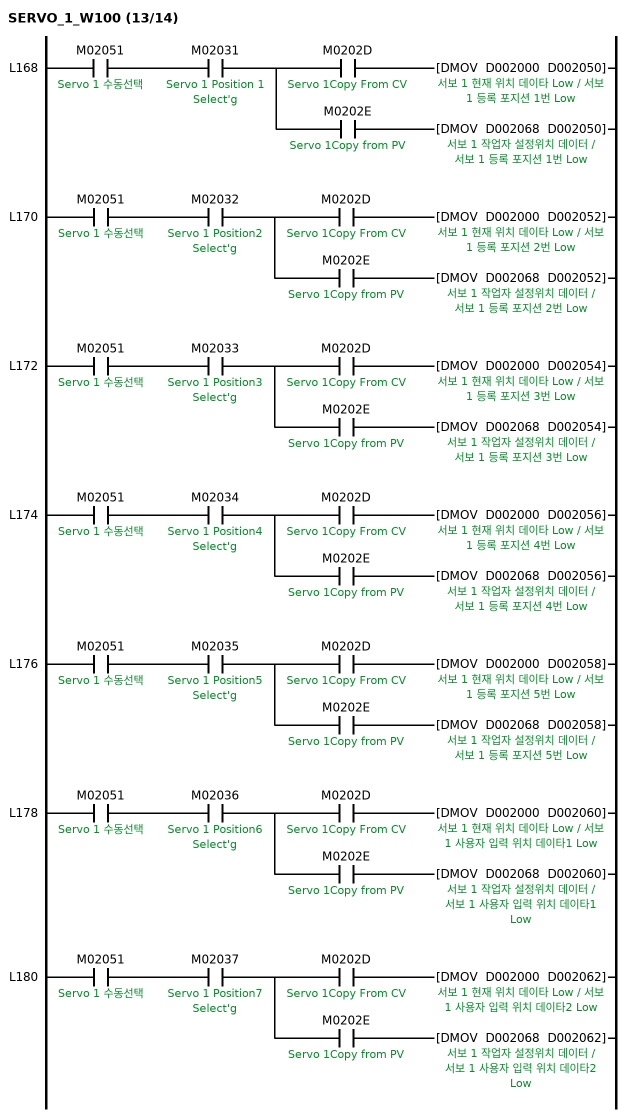
[picture p288: SERVO_1_W100 rungs L168-L180]
; L168
LOAD      M02051	// Servo 1 수동선택
AND       M02031	// Servo 1 Position 1 Select'g
MPUSH
AND       M0202D	// Servo 1Copy From CV
DMOV      D002000 D002050	// 서보 1 현재 위치 데이타 Low / 서보 1 등록 포지션 1번 Low
MPOP
AND       M0202E	// Servo 1Copy from PV
DMOV      D002068 D002050	// 서보 1 작업자 설정위치 데이터 / 서보 1 등록 포지션 1번 Low
; L170
LOAD      M02051	// Servo 1 수동선택
AND       M02032	// Servo 1 Position2 Select'g
MPUSH
AND       M0202D	// Servo 1Copy From CV
DMOV      D002000 D002052	// 서보 1 현재 위치 데이타 Low / 서보 1 등록 포지션 2번 Low
MPOP
AND       M0202E	// Servo 1Copy from PV
DMOV      D002068 D002052	// 서보 1 작업자 설정위치 데이터 / 서보 1 등록 포지션 2번 Low
; L172
LOAD      M02051	// Servo 1 수동선택
AND       M02033	// Servo 1 Position3 Select'g
MPUSH
AND       M0202D	// Servo 1Copy From CV
DMOV      D002000 D002054	// 서보 1 현재 위치 데이타 Low / 서보 1 등록 포지션 3번 Low
MPOP
AND       M0202E	// Servo 1Copy from PV
DMOV      D002068 D002054	// 서보 1 작업자 설정위치 데이터 / 서보 1 등록 포지션 3번 Low
; L174
LOAD      M02051	// Servo 1 수동선택
AND       M02034	// Servo 1 Position4 Select'g
MPUSH
AND       M0202D	// Servo 1Copy From CV
DMOV      D002000 D002056	// 서보 1 현재 위치 데이타 Low / 서보 1 등록 포지션 4번 Low
MPOP
AND       M0202E	// Servo 1Copy from PV
DMOV      D002068 D002056	// 서보 1 작업자 설정위치 데이터 / 서보 1 등록 포지션 4번 Low
; L176
LOAD      M02051	// Servo 1 수동선택
AND       M02035	// Servo 1 Position5 Select'g
MPUSH
AND       M0202D	// Servo 1Copy From CV
DMOV      D002000 D002058	// 서보 1 현재 위치 데이타 Low / 서보 1 등록 포지션 5번 Low
MPOP
AND       M0202E	// Servo 1Copy from PV
DMOV      D002068 D002058	// 서보 1 작업자 설정위치 데이터 / 서보 1 등록 포지션 5번 Low
; L178
LOAD      M02051	// Servo 1 수동선택
AND       M02036	// Servo 1 Position6 Select'g
MPUSH
AND       M0202D	// Servo 1Copy From CV
DMOV      D002000 D002060	// 서보 1 현재 위치 데이타 Low / 서보 1 사용자 입력 위치 데이타1 Low
MPOP
AND       M0202E	// Servo 1Copy from PV
DMOV      D002068 D002060	// 서보 1 작업자 설정위치 데이터 / 서보 1 사용자 입력 위치 데이타1 Low
; L180
LOAD      M02051	// Servo 1 수동선택
AND       M02037	// Servo 1 Position7 Select'g
MPUSH
AND       M0202D	// Servo 1Copy From CV
DMOV      D002000 D002062	// 서보 1 현재 위치 데이타 Low / 서보 1 사용자 입력 위치 데이타2 Low
MPOP
AND       M0202E	// Servo 1Copy from PV
DMOV      D002068 D002062	// 서보 1 작업자 설정위치 데이터 / 서보 1 사용자 입력 위치 데이타2 Low

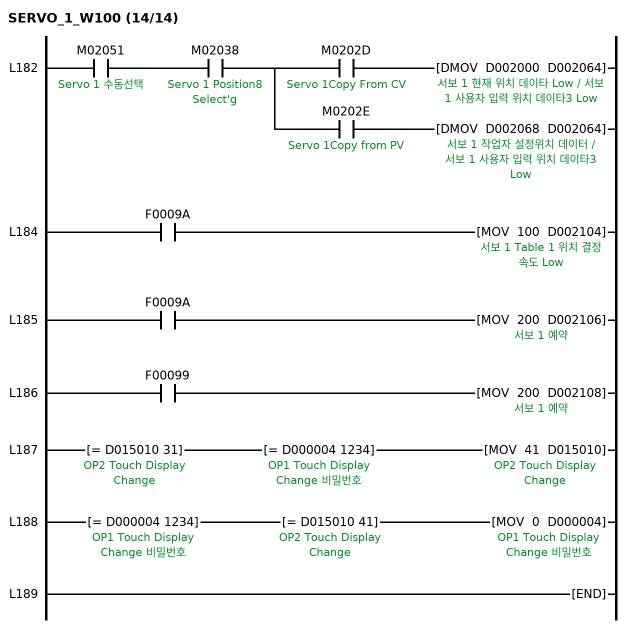
; L182
LOAD      M02051	// Servo 1 수동선택
AND       M02038	// Servo 1 Position8 Select'g
MPUSH
AND       M0202D	// Servo 1Copy From CV
DMOV      D002000 D002064	// 서보 1 현재 위치 데이타 Low / 서보 1 사용자 입력 위치 데이타3 Low
MPOP
AND       M0202E	// Servo 1Copy from PV
DMOV      D002068 D002064	// 서보 1 작업자 설정위치 데이터 / 서보 1 사용자 입력 위치 데이타3 Low
; L184
LOAD      F0009A
MOV       100 D002104	// 서보 1 Table 1 위치 결정 속도 Low
; L185
LOAD      F0009A
MOV       200 D002106	// 서보 1 예약
; L186
LOAD      F00099
MOV       200 D002108	// 서보 1 예약
; L187
LOAD=     D015010 31	// OP2 Touch Display Change
AND=      D000004 1234	// OP1 Touch Display Change 비밀번호
MOV       41 D015010	// OP2 Touch Display Change
; L188
LOAD=     D000004 1234	// OP1 Touch Display Change 비밀번호
AND=      D015010 41	// OP2 Touch Display Change
MOV       0 D000004	// OP1 Touch Display Change 비밀번호
; L189
END

PROGRAM SERVO_2_W200 (task: 스캔 프로그램)

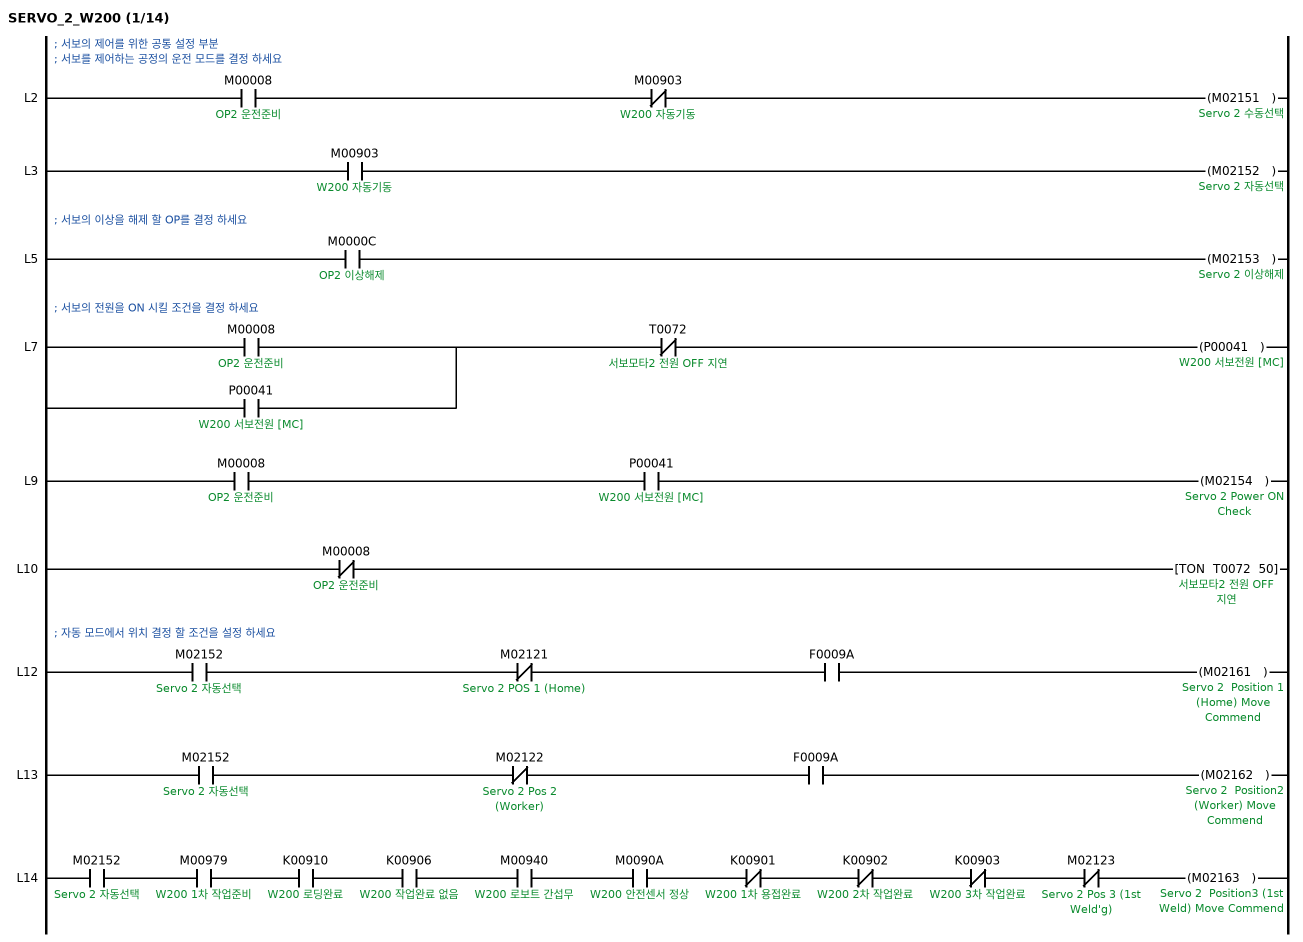
// 서보의 제어를 위한 공통 설정 부분
//     서보를 제어하는 공정의 운전 모드를 결정 하세요
; L2
LOAD      M00008	// OP2 운전준비
AND NOT   M00903	// W200 자동기동
OUT       M02151	// Servo 2 수동선택
; L3
LOAD      M00903	// W200 자동기동
OUT       M02152	// Servo 2 자동선택
//     서보의 이상을 해제 할 OP를 결정 하세요
; L5
LOAD      M0000C	// OP2 이상해제
OUT       M02153	// Servo 2 이상해제
//     서보의 전원을 ON 시킬 조건을 결정 하세요
; L7
LOAD      M00008	// OP2 운전준비
OR        P00041	// W200 서보전원 [MC]
AND NOT   T0072	// 서보모타2 전원 OFF 지연
OUT       P00041	// W200 서보전원 [MC]
; L9
LOAD      M00008	// OP2 운전준비
AND       P00041	// W200 서보전원 [MC]
OUT       M02154	// Servo 2 Power ON Check
; L10
LOAD NOT  M00008	// OP2 운전준비
TON       T0072 50	// 서보모타2 전원 OFF 지연
//     자동 모드에서 위치 결정 할 조건을 설정 하세요
; L12
LOAD      M02152	// Servo 2 자동선택
AND NOT   M02121	// Servo 2 POS 1 (Home)
AND       F0009A
OUT       M02161	// Servo 2  Position 1 (Home) Move Commend
; L13
LOAD      M02152	// Servo 2 자동선택
AND NOT   M02122	// Servo 2 Pos 2 (Worker)
AND       F0009A
OUT       M02162	// Servo 2  Position2 (Worker) Move Commend
; L14
LOAD      M02152	// Servo 2 자동선택
AND       M00979	// W200 1차 작업준비
AND       K00910	// W200 로딩완료
AND       K00906	// W200 작업완료 없음
AND       M00940	// W200 로보트 간섭무
AND       M0090A	// W200 안전센서 정상
AND NOT   K00901	// W200 1차 용접완료
AND NOT   K00902	// W200 2차 작업완료
AND NOT   K00903	// W200 3차 작업완료
AND NOT   M02123	// Servo 2 Pos 3 (1st Weld'g)
OUT       M02163	// Servo 2  Position3 (1st Weld) Move Commend

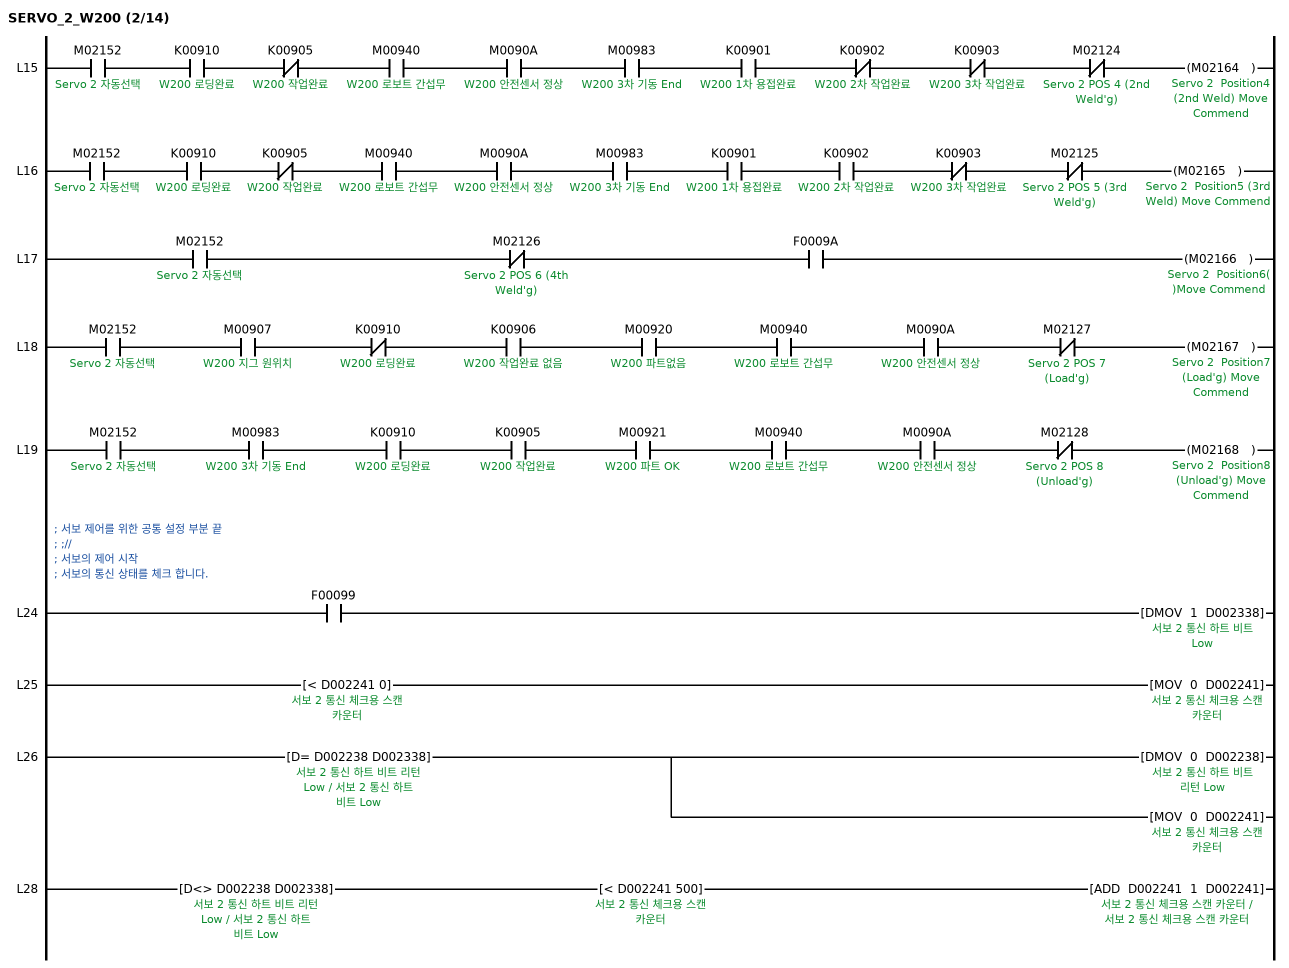
; L15
LOAD      M02152	// Servo 2 자동선택
AND       K00910	// W200 로딩완료
AND NOT   K00905	// W200 작업완료
AND       M00940	// W200 로보트 간섭무
AND       M0090A	// W200 안전센서 정상
AND       M00983	// W200 3차 기동 End
AND       K00901	// W200 1차 용접완료
AND NOT   K00902	// W200 2차 작업완료
AND NOT   K00903	// W200 3차 작업완료
AND NOT   M02124	// Servo 2 POS 4 (2nd Weld'g)
OUT       M02164	// Servo 2  Position4 (2nd Weld) Move Commend
; L16
LOAD      M02152	// Servo 2 자동선택
AND       K00910	// W200 로딩완료
AND NOT   K00905	// W200 작업완료
AND       M00940	// W200 로보트 간섭무
AND       M0090A	// W200 안전센서 정상
AND       M00983	// W200 3차 기동 End
AND       K00901	// W200 1차 용접완료
AND       K00902	// W200 2차 작업완료
AND NOT   K00903	// W200 3차 작업완료
AND NOT   M02125	// Servo 2 POS 5 (3rd Weld'g)
OUT       M02165	// Servo 2  Position5 (3rd Weld) Move Commend
; L17
LOAD      M02152	// Servo 2 자동선택
AND NOT   M02126	// Servo 2 POS 6 (4th Weld'g)
AND       F0009A
OUT       M02166	// Servo 2  Position6()Move Commend
; L18
LOAD      M02152	// Servo 2 자동선택
AND       M00907	// W200 지그 원위치
AND NOT   K00910	// W200 로딩완료
AND       K00906	// W200 작업완료 없음
AND       M00920	// W200 파트없음
AND       M00940	// W200 로보트 간섭무
AND       M0090A	// W200 안전센서 정상
AND NOT   M02127	// Servo 2 POS 7 (Load'g)
OUT       M02167	// Servo 2  Position7 (Load'g) Move Commend
; L19
LOAD      M02152	// Servo 2 자동선택
AND       M00983	// W200 3차 기동 End
AND       K00910	// W200 로딩완료
AND       K00905	// W200 작업완료
AND       M00921	// W200 파트 OK
AND       M00940	// W200 로보트 간섭무
AND       M0090A	// W200 안전센서 정상
AND NOT   M02128	// Servo 2 POS 8 (Unload'g)
OUT       M02168	// Servo 2  Position8 (Unload'g) Move Commend
// 서보 제어를 위한 공통 설정 부분 끝
// ;//
// 서보의 제어 시작
//     서보의 통신 상태를 체크 합니다.
; L24
LOAD      F00099
DMOV      1 D002338	// 서보 2 통신 하트 비트 Low
; L25
LOAD<     D002241 0	// 서보 2 통신 체크용 스캔 카운터
MOV       0 D002241	// 서보 2 통신 체크용 스캔 카운터
; L26
LOADD=    D002238 D002338	// 서보 2 통신 하트 비트 리턴 Low / 서보 2 통신 하트 비트 Low
DMOV      0 D002238	// 서보 2 통신 하트 비트 리턴 Low
MOV       0 D002241	// 서보 2 통신 체크용 스캔 카운터
; L28
LOADD<>   D002238 D002338	// 서보 2 통신 하트 비트 리턴 Low / 서보 2 통신 하트 비트 Low
AND<      D002241 500	// 서보 2 통신 체크용 스캔 카운터
ADD       D002241 1 D002241	// 서보 2 통신 체크용 스캔 카운터 / 서보 2 통신 체크용 스캔 카운터

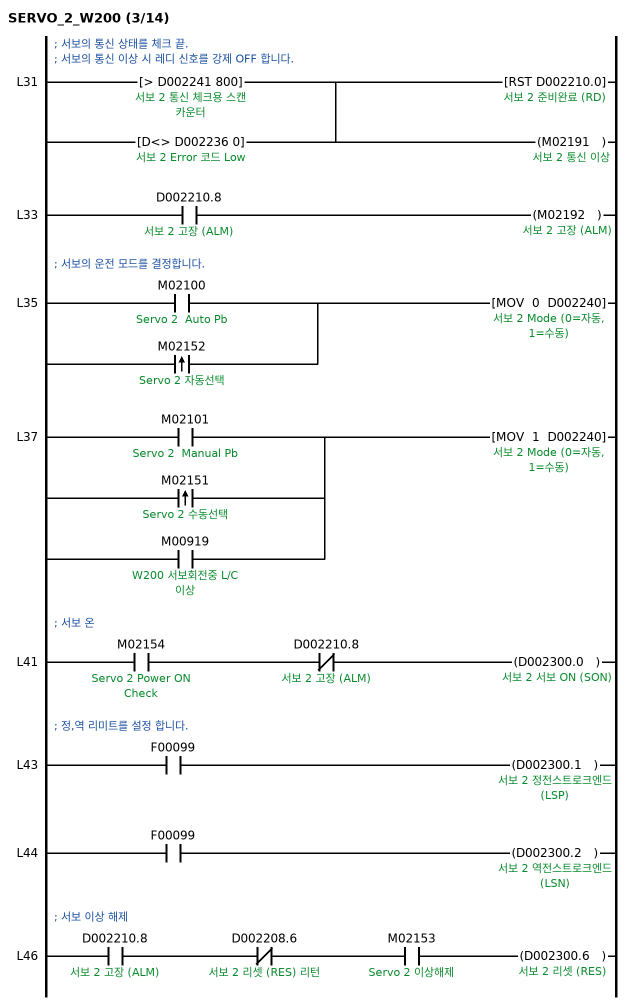
//     서보의 통신 상태를 체크 끝.
//     서보의 통신 이상 시 레디 신호를 강제 OFF 합니다.
; L31
LOAD>     D002241 800	// 서보 2 통신 체크용 스캔 카운터
ORD<>     D002236 0	// 서보 2 Error 코드 Low
RST       D002210.0	// 서보 2 준비완료 (RD)
OUT       M02191	// 서보 2 통신 이상
; L33
LOAD      D002210.8	// 서보 2 고장 (ALM)
OUT       M02192	// 서보 2 고장 (ALM)
//     서보의 운전 모드를 결정합니다.
; L35
LOAD      M02100	// Servo 2  Auto Pb
ORP       M02152	// Servo 2 자동선택
MOV       0 D002240	// 서보 2 Mode (0=자동, 1=수동)
; L37
LOAD      M02101	// Servo 2  Manual Pb
ORP       M02151	// Servo 2 수동선택
OR        M00919	// W200 서보회전중 L/C 이상
MOV       1 D002240	// 서보 2 Mode (0=자동, 1=수동)
//     서보 온
; L41
LOAD      M02154	// Servo 2 Power ON Check
AND NOT   D002210.8	// 서보 2 고장 (ALM)
OUT       D002300.0	// 서보 2 서보 ON (SON)
//     정,역 리미트를 설정 합니다.
; L43
LOAD      F00099
OUT       D002300.1	// 서보 2 정전스트로크엔드 (LSP)
; L44
LOAD      F00099
OUT       D002300.2	// 서보 2 역전스트로크엔드 (LSN)
//     서보 이상 해제
; L46
LOAD      D002210.8	// 서보 2 고장 (ALM)
AND NOT   D002208.6	// 서보 2 리셋 (RES) 리턴
AND       M02153	// Servo 2 이상해제
OUT       D002300.6	// 서보 2 리셋 (RES)

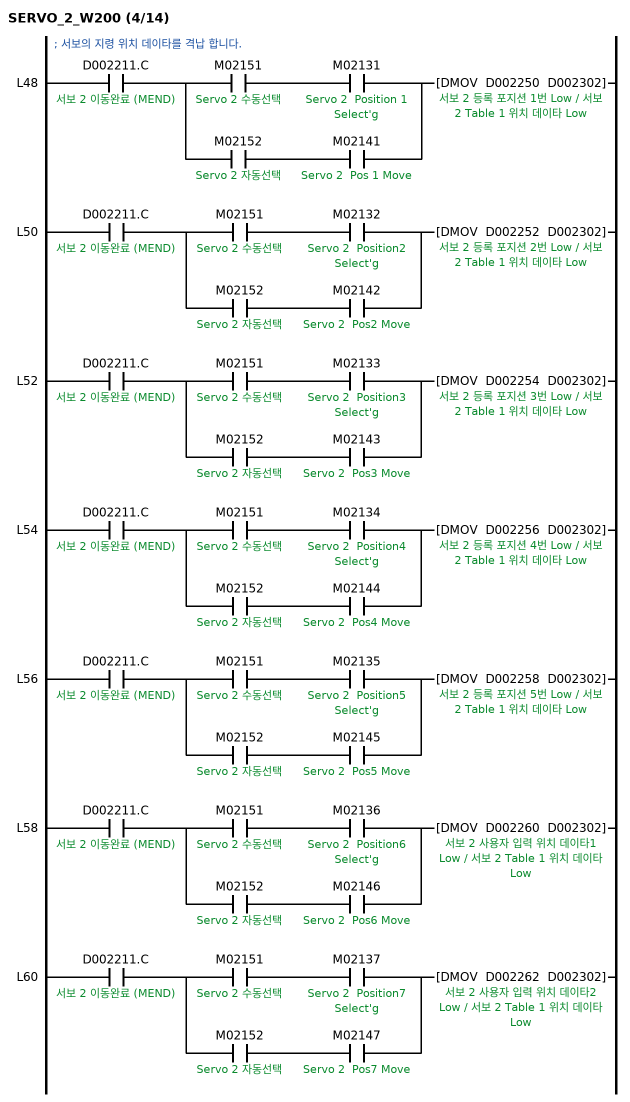
//     서보의 지령 위치 데이타를 격납 합니다.
; L48
LOAD      D002211.C	// 서보 2 이동완료 (MEND)
LOAD      M02151	// Servo 2 수동선택
AND       M02131	// Servo 2  Position 1 Select'g
LOAD      M02152	// Servo 2 자동선택
AND       M02141	// Servo 2  Pos 1 Move
OR LOAD
AND LOAD
DMOV      D002250 D002302	// 서보 2 등록 포지션 1번 Low / 서보 2 Table 1 위치 데이타 Low
; L50
LOAD      D002211.C	// 서보 2 이동완료 (MEND)
LOAD      M02151	// Servo 2 수동선택
AND       M02132	// Servo 2  Position2 Select'g
LOAD      M02152	// Servo 2 자동선택
AND       M02142	// Servo 2  Pos2 Move
OR LOAD
AND LOAD
DMOV      D002252 D002302	// 서보 2 등록 포지션 2번 Low / 서보 2 Table 1 위치 데이타 Low
; L52
LOAD      D002211.C	// 서보 2 이동완료 (MEND)
LOAD      M02151	// Servo 2 수동선택
AND       M02133	// Servo 2  Position3 Select'g
LOAD      M02152	// Servo 2 자동선택
AND       M02143	// Servo 2  Pos3 Move
OR LOAD
AND LOAD
DMOV      D002254 D002302	// 서보 2 등록 포지션 3번 Low / 서보 2 Table 1 위치 데이타 Low
; L54
LOAD      D002211.C	// 서보 2 이동완료 (MEND)
LOAD      M02151	// Servo 2 수동선택
AND       M02134	// Servo 2  Position4 Select'g
LOAD      M02152	// Servo 2 자동선택
AND       M02144	// Servo 2  Pos4 Move
OR LOAD
AND LOAD
DMOV      D002256 D002302	// 서보 2 등록 포지션 4번 Low / 서보 2 Table 1 위치 데이타 Low
; L56
LOAD      D002211.C	// 서보 2 이동완료 (MEND)
LOAD      M02151	// Servo 2 수동선택
AND       M02135	// Servo 2  Position5 Select'g
LOAD      M02152	// Servo 2 자동선택
AND       M02145	// Servo 2  Pos5 Move
OR LOAD
AND LOAD
DMOV      D002258 D002302	// 서보 2 등록 포지션 5번 Low / 서보 2 Table 1 위치 데이타 Low
; L58
LOAD      D002211.C	// 서보 2 이동완료 (MEND)
LOAD      M02151	// Servo 2 수동선택
AND       M02136	// Servo 2  Position6 Select'g
LOAD      M02152	// Servo 2 자동선택
AND       M02146	// Servo 2  Pos6 Move
OR LOAD
AND LOAD
DMOV      D002260 D002302	// 서보 2 사용자 입력 위치 데이타1 Low / 서보 2 Table 1 위치 데이타 Low
; L60
LOAD      D002211.C	// 서보 2 이동완료 (MEND)
LOAD      M02151	// Servo 2 수동선택
AND       M02137	// Servo 2  Position7 Select'g
LOAD      M02152	// Servo 2 자동선택
AND       M02147	// Servo 2  Pos7 Move
OR LOAD
AND LOAD
DMOV      D002262 D002302	// 서보 2 사용자 입력 위치 데이타2 Low / 서보 2 Table 1 위치 데이타 Low

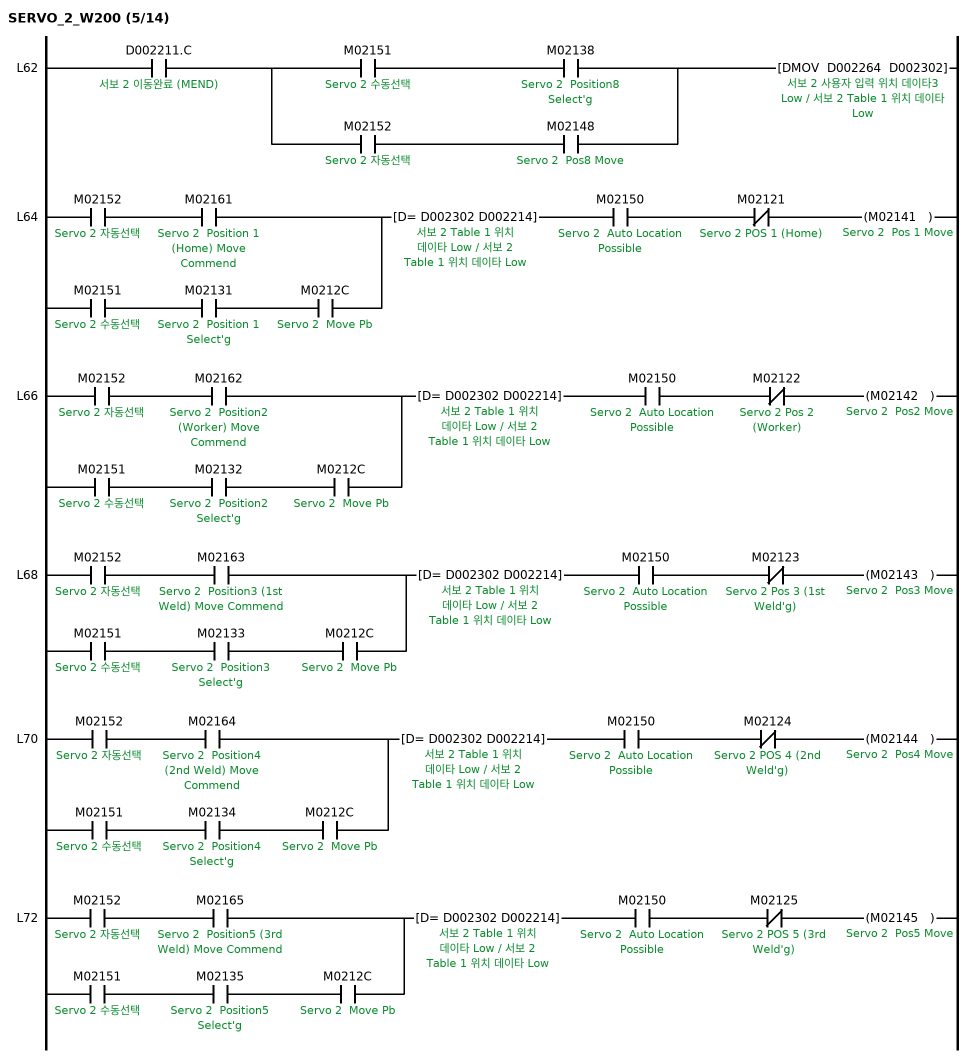
; L62
LOAD      D002211.C	// 서보 2 이동완료 (MEND)
LOAD      M02151	// Servo 2 수동선택
AND       M02138	// Servo 2  Position8 Select'g
LOAD      M02152	// Servo 2 자동선택
AND       M02148	// Servo 2  Pos8 Move
OR LOAD
AND LOAD
DMOV      D002264 D002302	// 서보 2 사용자 입력 위치 데이타3 Low / 서보 2 Table 1 위치 데이타 Low
; L64
LOAD      M02152	// Servo 2 자동선택
AND       M02161	// Servo 2  Position 1 (Home) Move Commend
LOAD      M02151	// Servo 2 수동선택
AND       M02131	// Servo 2  Position 1 Select'g
AND       M0212C	// Servo 2  Move Pb
OR LOAD
ANDD=     D002302 D002214	// 서보 2 Table 1 위치 데이타 Low / 서보 2 Table 1 위치 데이타 Low
AND       M02150	// Servo 2  Auto Location Possible
AND NOT   M02121	// Servo 2 POS 1 (Home)
OUT       M02141	// Servo 2  Pos 1 Move
; L66
LOAD      M02152	// Servo 2 자동선택
AND       M02162	// Servo 2  Position2 (Worker) Move Commend
LOAD      M02151	// Servo 2 수동선택
AND       M02132	// Servo 2  Position2 Select'g
AND       M0212C	// Servo 2  Move Pb
OR LOAD
ANDD=     D002302 D002214	// 서보 2 Table 1 위치 데이타 Low / 서보 2 Table 1 위치 데이타 Low
AND       M02150	// Servo 2  Auto Location Possible
AND NOT   M02122	// Servo 2 Pos 2 (Worker)
OUT       M02142	// Servo 2  Pos2 Move
; L68
LOAD      M02152	// Servo 2 자동선택
AND       M02163	// Servo 2  Position3 (1st Weld) Move Commend
LOAD      M02151	// Servo 2 수동선택
AND       M02133	// Servo 2  Position3 Select'g
AND       M0212C	// Servo 2  Move Pb
OR LOAD
ANDD=     D002302 D002214	// 서보 2 Table 1 위치 데이타 Low / 서보 2 Table 1 위치 데이타 Low
AND       M02150	// Servo 2  Auto Location Possible
AND NOT   M02123	// Servo 2 Pos 3 (1st Weld'g)
OUT       M02143	// Servo 2  Pos3 Move
; L70
LOAD      M02152	// Servo 2 자동선택
AND       M02164	// Servo 2  Position4 (2nd Weld) Move Commend
LOAD      M02151	// Servo 2 수동선택
AND       M02134	// Servo 2  Position4 Select'g
AND       M0212C	// Servo 2  Move Pb
OR LOAD
ANDD=     D002302 D002214	// 서보 2 Table 1 위치 데이타 Low / 서보 2 Table 1 위치 데이타 Low
AND       M02150	// Servo 2  Auto Location Possible
AND NOT   M02124	// Servo 2 POS 4 (2nd Weld'g)
OUT       M02144	// Servo 2  Pos4 Move
; L72
LOAD      M02152	// Servo 2 자동선택
AND       M02165	// Servo 2  Position5 (3rd Weld) Move Commend
LOAD      M02151	// Servo 2 수동선택
AND       M02135	// Servo 2  Position5 Select'g
AND       M0212C	// Servo 2  Move Pb
OR LOAD
ANDD=     D002302 D002214	// 서보 2 Table 1 위치 데이타 Low / 서보 2 Table 1 위치 데이타 Low
AND       M02150	// Servo 2  Auto Location Possible
AND NOT   M02125	// Servo 2 POS 5 (3rd Weld'g)
OUT       M02145	// Servo 2  Pos5 Move

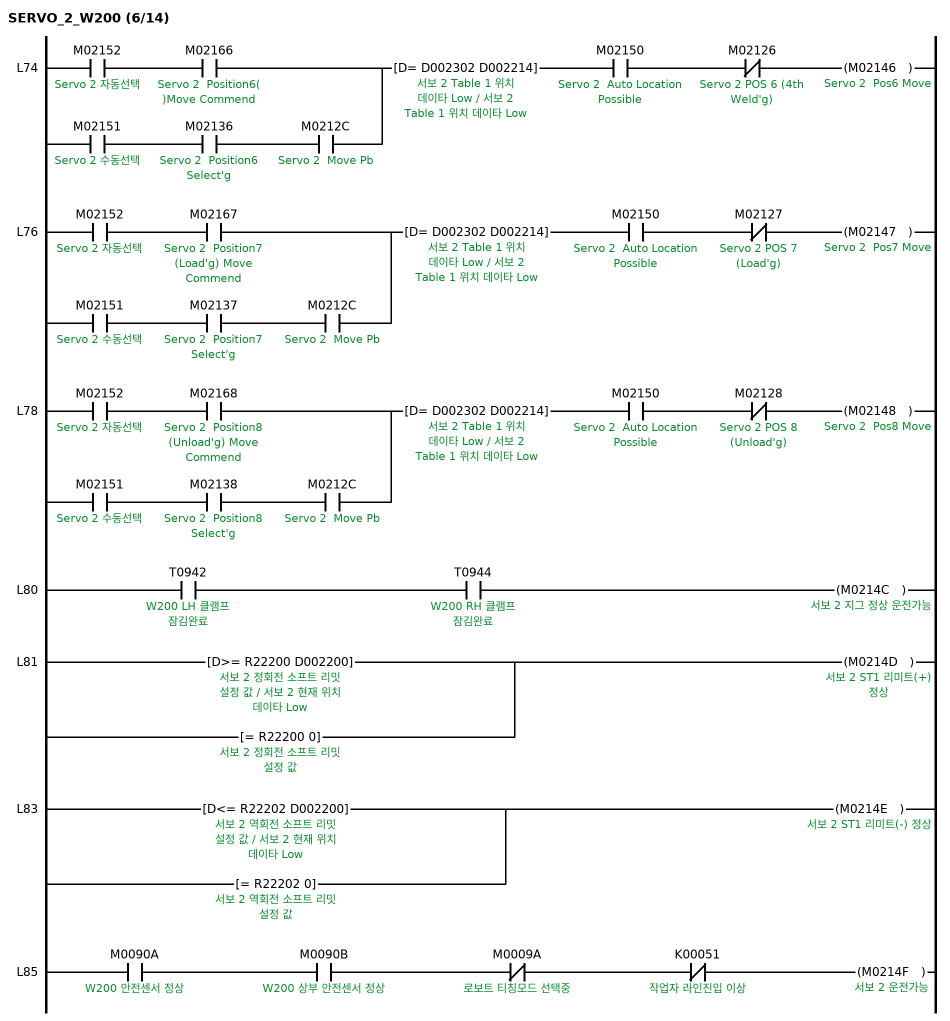
; L74
LOAD      M02152	// Servo 2 자동선택
AND       M02166	// Servo 2  Position6()Move Commend
LOAD      M02151	// Servo 2 수동선택
AND       M02136	// Servo 2  Position6 Select'g
AND       M0212C	// Servo 2  Move Pb
OR LOAD
ANDD=     D002302 D002214	// 서보 2 Table 1 위치 데이타 Low / 서보 2 Table 1 위치 데이타 Low
AND       M02150	// Servo 2  Auto Location Possible
AND NOT   M02126	// Servo 2 POS 6 (4th Weld'g)
OUT       M02146	// Servo 2  Pos6 Move
; L76
LOAD      M02152	// Servo 2 자동선택
AND       M02167	// Servo 2  Position7 (Load'g) Move Commend
LOAD      M02151	// Servo 2 수동선택
AND       M02137	// Servo 2  Position7 Select'g
AND       M0212C	// Servo 2  Move Pb
OR LOAD
ANDD=     D002302 D002214	// 서보 2 Table 1 위치 데이타 Low / 서보 2 Table 1 위치 데이타 Low
AND       M02150	// Servo 2  Auto Location Possible
AND NOT   M02127	// Servo 2 POS 7 (Load'g)
OUT       M02147	// Servo 2  Pos7 Move
; L78
LOAD      M02152	// Servo 2 자동선택
AND       M02168	// Servo 2  Position8 (Unload'g) Move Commend
LOAD      M02151	// Servo 2 수동선택
AND       M02138	// Servo 2  Position8 Select'g
AND       M0212C	// Servo 2  Move Pb
OR LOAD
ANDD=     D002302 D002214	// 서보 2 Table 1 위치 데이타 Low / 서보 2 Table 1 위치 데이타 Low
AND       M02150	// Servo 2  Auto Location Possible
AND NOT   M02128	// Servo 2 POS 8 (Unload'g)
OUT       M02148	// Servo 2  Pos8 Move
; L80
LOAD      T0942	// W200 LH 클램프 잠김완료
AND       T0944	// W200 RH 클램프 잠김완료
OUT       M0214C	// 서보 2 지그 정상 운전가능
; L81
LOADD>=   R22200 D002200	// 서보 2 정회전 소프트 리밋 설정 값 / 서보 2 현재 위치 데이타 Low
OR=       R22200 0	// 서보 2 정회전 소프트 리밋 설정 값
OUT       M0214D	// 서보 2 ST1 리미트(+) 정상
; L83
LOADD<=   R22202 D002200	// 서보 2 역회전 소프트 리밋 설정 값 / 서보 2 현재 위치 데이타 Low
OR=       R22202 0	// 서보 2 역회전 소프트 리밋 설정 값
OUT       M0214E	// 서보 2 ST1 리미트(-) 정상
; L85
LOAD      M0090A	// W200 안전센서 정상
AND       M0090B	// W200 상부 안전센서 정상
AND NOT   M0009A	// 로보트 티칭모드 선택중
AND NOT   K00051	//  작업자 라인진입 이상
OUT       M0214F	// 서보 2 운전가능

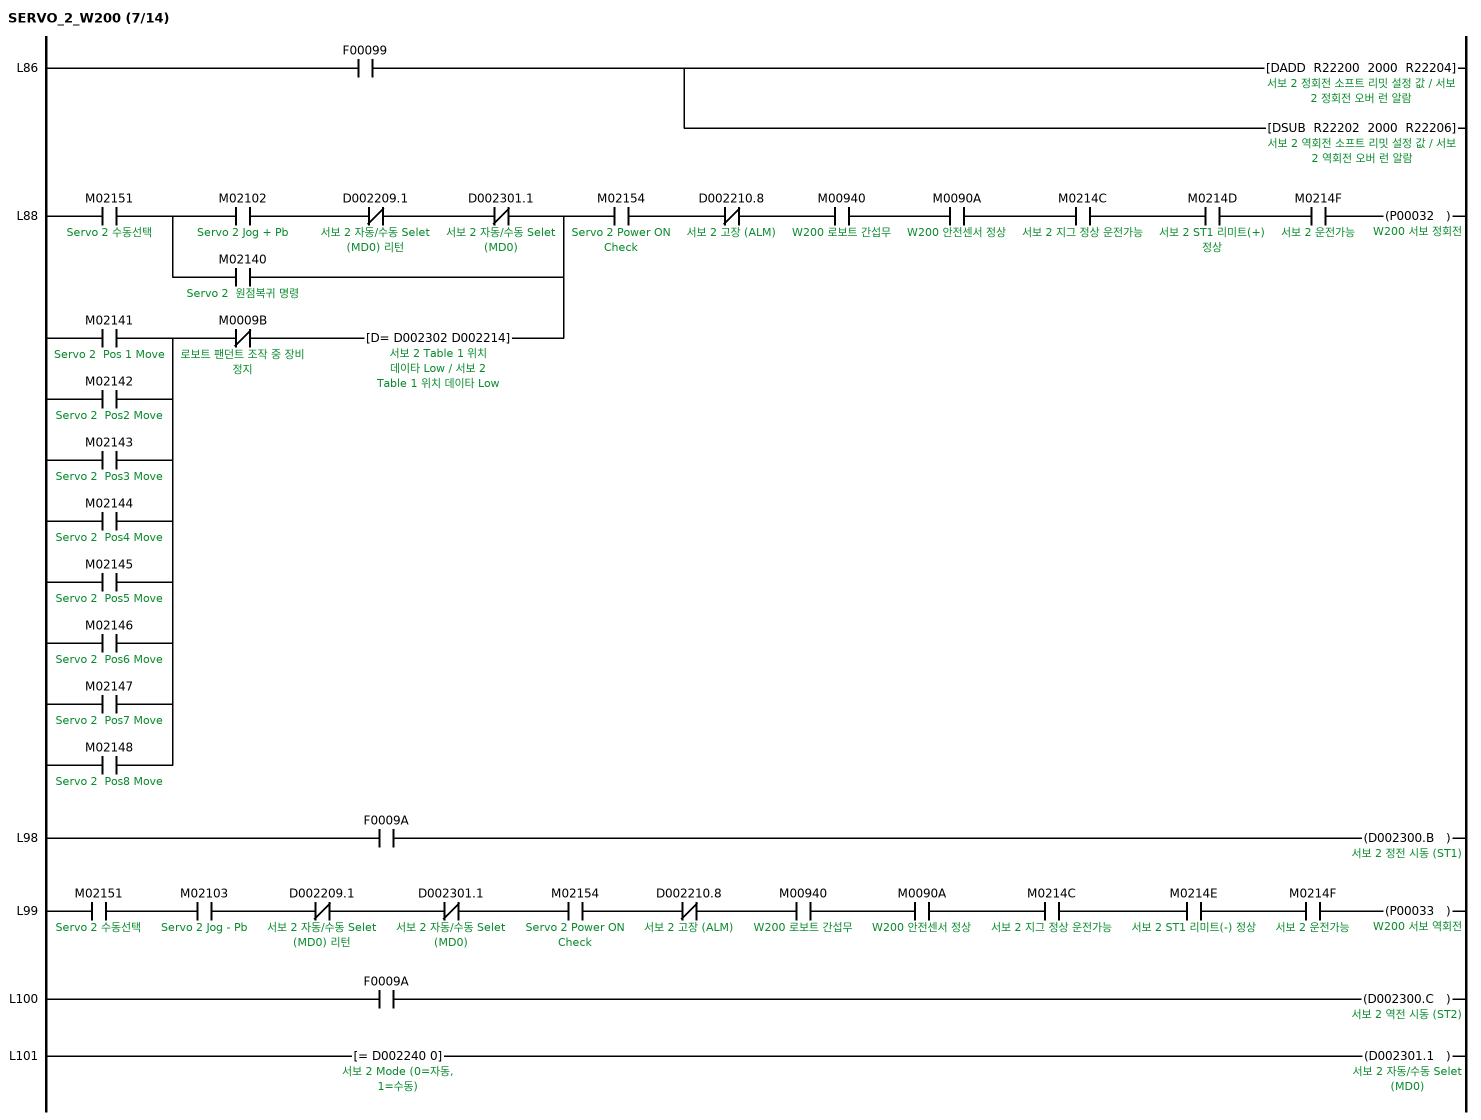
; L86
LOAD      F00099
DADD      R22200 2000 R22204	// 서보 2 정회전 소프트 리밋 설정 값 / 서보 2 정회전 오버 런 알람
DSUB      R22202 2000 R22206	// 서보 2 역회전 소프트 리밋 설정 값 / 서보 2 역회전 오버 런 알람
; L88
LOAD      M02151	// Servo 2 수동선택
LOAD      M02102	// Servo 2 Jog + Pb
AND NOT   D002209.1	// 서보 2 자동/수동 Selet (MD0) 리턴
AND NOT   D002301.1	// 서보 2 자동/수동 Selet (MD0)
OR        M02140	// Servo 2  원점복귀 명령
AND LOAD
LOAD      M02141	// Servo 2  Pos 1 Move
OR        M02142	// Servo 2  Pos2 Move
OR        M02143	// Servo 2  Pos3 Move
OR        M02144	// Servo 2  Pos4 Move
OR        M02145	// Servo 2  Pos5 Move
OR        M02146	// Servo 2  Pos6 Move
OR        M02147	// Servo 2  Pos7 Move
OR        M02148	// Servo 2  Pos8 Move
AND NOT   M0009B	// 로보트 팬던트 조작 중 장비 정지
ANDD=     D002302 D002214	// 서보 2 Table 1 위치 데이타 Low / 서보 2 Table 1 위치 데이타 Low
OR LOAD
AND       M02154	// Servo 2 Power ON Check
AND NOT   D002210.8	// 서보 2 고장 (ALM)
AND       M00940	// W200 로보트 간섭무
AND       M0090A	// W200 안전센서 정상
AND       M0214C	// 서보 2 지그 정상 운전가능
AND       M0214D	// 서보 2 ST1 리미트(+) 정상
AND       M0214F	// 서보 2 운전가능
OUT       P00032	// W200 서보 정회전
; L98
LOAD      F0009A
OUT       D002300.B	// 서보 2 정전 시동 (ST1)
; L99
LOAD      M02151	// Servo 2 수동선택
AND       M02103	// Servo 2 Jog - Pb
AND NOT   D002209.1	// 서보 2 자동/수동 Selet (MD0) 리턴
AND NOT   D002301.1	// 서보 2 자동/수동 Selet (MD0)
AND       M02154	// Servo 2 Power ON Check
AND NOT   D002210.8	// 서보 2 고장 (ALM)
AND       M00940	// W200 로보트 간섭무
AND       M0090A	// W200 안전센서 정상
AND       M0214C	// 서보 2 지그 정상 운전가능
AND       M0214E	// 서보 2 ST1 리미트(-) 정상
AND       M0214F	// 서보 2 운전가능
OUT       P00033	// W200 서보 역회전
; L100
LOAD      F0009A
OUT       D002300.C	// 서보 2 역전 시동 (ST2)
; L101
LOAD=     D002240 0	// 서보 2 Mode (0=자동, 1=수동)
OUT       D002301.1	// 서보 2 자동/수동 Selet (MD0)

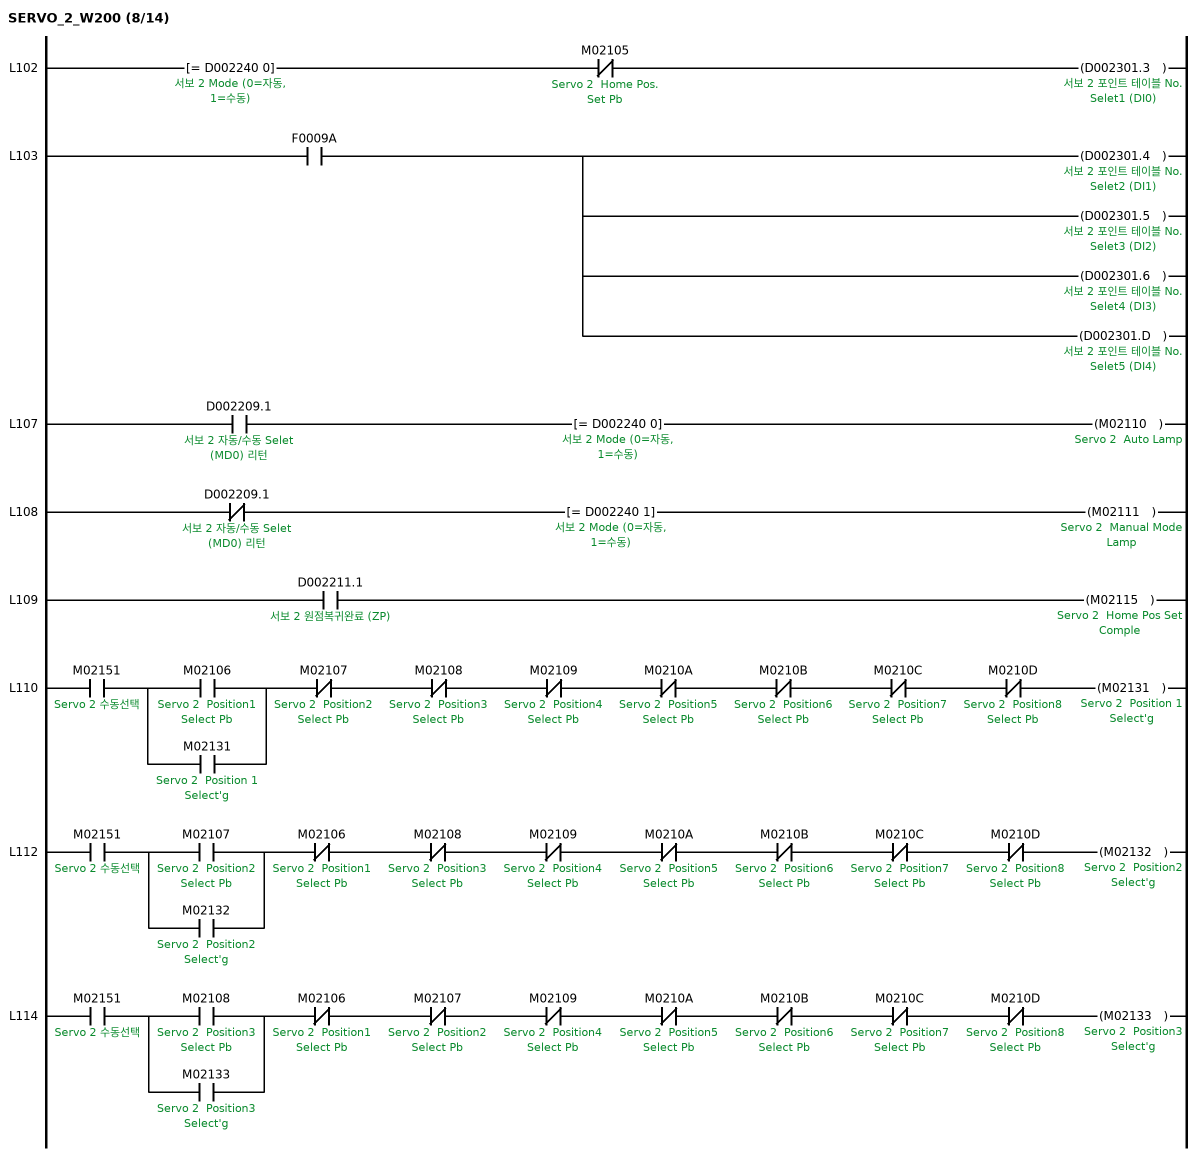
; L102
LOAD=     D002240 0	// 서보 2 Mode (0=자동, 1=수동)
AND NOT   M02105	// Servo 2  Home Pos. Set Pb
OUT       D002301.3	// 서보 2 포인트 테이블 No. Selet1 (DI0)
; L103
LOAD      F0009A
OUT       D002301.4	// 서보 2 포인트 테이블 No. Selet2 (DI1)
OUT       D002301.5	// 서보 2 포인트 테이블 No. Selet3 (DI2)
OUT       D002301.6	// 서보 2 포인트 테이블 No. Selet4 (DI3)
OUT       D002301.D	// 서보 2 포인트 테이블 No. Selet5 (DI4)
; L107
LOAD      D002209.1	// 서보 2 자동/수동 Selet (MD0) 리턴
AND=      D002240 0	// 서보 2 Mode (0=자동, 1=수동)
OUT       M02110	// Servo 2  Auto Lamp
; L108
LOAD NOT  D002209.1	// 서보 2 자동/수동 Selet (MD0) 리턴
AND=      D002240 1	// 서보 2 Mode (0=자동, 1=수동)
OUT       M02111	// Servo 2  Manual Mode Lamp
; L109
LOAD      D002211.1	// 서보 2 원점복귀완료 (ZP)
OUT       M02115	// Servo 2  Home Pos Set Comple
; L110
LOAD      M02151	// Servo 2 수동선택
LOAD      M02106	// Servo 2  Position1 Select Pb
OR        M02131	// Servo 2  Position 1 Select'g
AND LOAD
AND NOT   M02107	// Servo 2  Position2 Select Pb
AND NOT   M02108	// Servo 2  Position3 Select Pb
AND NOT   M02109	// Servo 2  Position4 Select Pb
AND NOT   M0210A	// Servo 2  Position5 Select Pb
AND NOT   M0210B	// Servo 2  Position6 Select Pb
AND NOT   M0210C	// Servo 2  Position7 Select Pb
AND NOT   M0210D	// Servo 2  Position8 Select Pb
OUT       M02131	// Servo 2  Position 1 Select'g
; L112
LOAD      M02151	// Servo 2 수동선택
LOAD      M02107	// Servo 2  Position2 Select Pb
OR        M02132	// Servo 2  Position2 Select'g
AND LOAD
AND NOT   M02106	// Servo 2  Position1 Select Pb
AND NOT   M02108	// Servo 2  Position3 Select Pb
AND NOT   M02109	// Servo 2  Position4 Select Pb
AND NOT   M0210A	// Servo 2  Position5 Select Pb
AND NOT   M0210B	// Servo 2  Position6 Select Pb
AND NOT   M0210C	// Servo 2  Position7 Select Pb
AND NOT   M0210D	// Servo 2  Position8 Select Pb
OUT       M02132	// Servo 2  Position2 Select'g
; L114
LOAD      M02151	// Servo 2 수동선택
LOAD      M02108	// Servo 2  Position3 Select Pb
OR        M02133	// Servo 2  Position3 Select'g
AND LOAD
AND NOT   M02106	// Servo 2  Position1 Select Pb
AND NOT   M02107	// Servo 2  Position2 Select Pb
AND NOT   M02109	// Servo 2  Position4 Select Pb
AND NOT   M0210A	// Servo 2  Position5 Select Pb
AND NOT   M0210B	// Servo 2  Position6 Select Pb
AND NOT   M0210C	// Servo 2  Position7 Select Pb
AND NOT   M0210D	// Servo 2  Position8 Select Pb
OUT       M02133	// Servo 2  Position3 Select'g

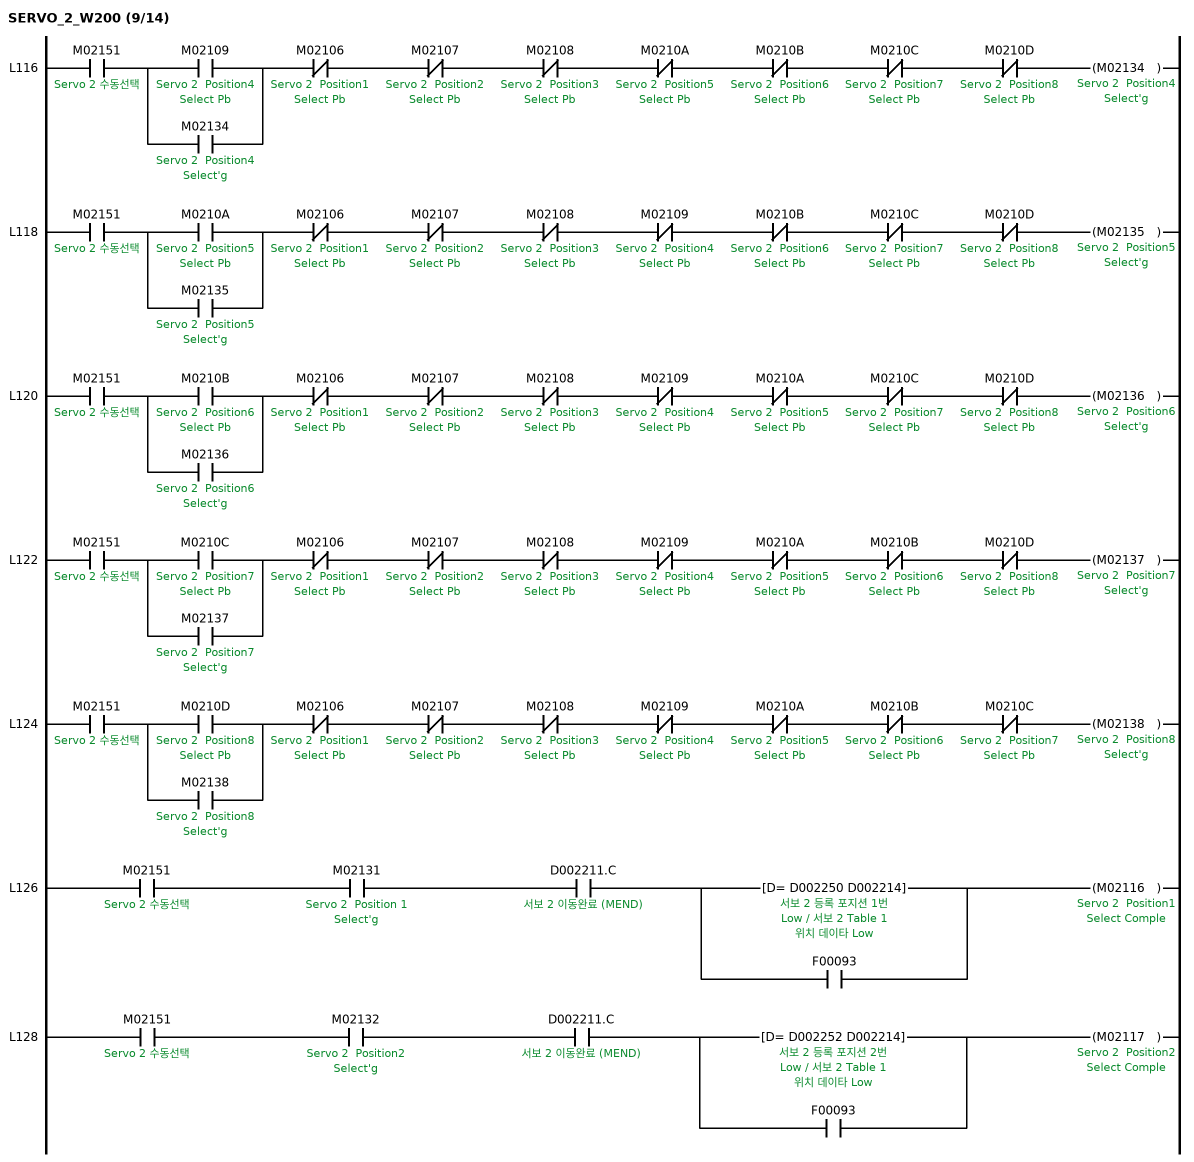
; L116
LOAD      M02151	// Servo 2 수동선택
LOAD      M02109	// Servo 2  Position4 Select Pb
OR        M02134	// Servo 2  Position4 Select'g
AND LOAD
AND NOT   M02106	// Servo 2  Position1 Select Pb
AND NOT   M02107	// Servo 2  Position2 Select Pb
AND NOT   M02108	// Servo 2  Position3 Select Pb
AND NOT   M0210A	// Servo 2  Position5 Select Pb
AND NOT   M0210B	// Servo 2  Position6 Select Pb
AND NOT   M0210C	// Servo 2  Position7 Select Pb
AND NOT   M0210D	// Servo 2  Position8 Select Pb
OUT       M02134	// Servo 2  Position4 Select'g
; L118
LOAD      M02151	// Servo 2 수동선택
LOAD      M0210A	// Servo 2  Position5 Select Pb
OR        M02135	// Servo 2  Position5 Select'g
AND LOAD
AND NOT   M02106	// Servo 2  Position1 Select Pb
AND NOT   M02107	// Servo 2  Position2 Select Pb
AND NOT   M02108	// Servo 2  Position3 Select Pb
AND NOT   M02109	// Servo 2  Position4 Select Pb
AND NOT   M0210B	// Servo 2  Position6 Select Pb
AND NOT   M0210C	// Servo 2  Position7 Select Pb
AND NOT   M0210D	// Servo 2  Position8 Select Pb
OUT       M02135	// Servo 2  Position5 Select'g
; L120
LOAD      M02151	// Servo 2 수동선택
LOAD      M0210B	// Servo 2  Position6 Select Pb
OR        M02136	// Servo 2  Position6 Select'g
AND LOAD
AND NOT   M02106	// Servo 2  Position1 Select Pb
AND NOT   M02107	// Servo 2  Position2 Select Pb
AND NOT   M02108	// Servo 2  Position3 Select Pb
AND NOT   M02109	// Servo 2  Position4 Select Pb
AND NOT   M0210A	// Servo 2  Position5 Select Pb
AND NOT   M0210C	// Servo 2  Position7 Select Pb
AND NOT   M0210D	// Servo 2  Position8 Select Pb
OUT       M02136	// Servo 2  Position6 Select'g
; L122
LOAD      M02151	// Servo 2 수동선택
LOAD      M0210C	// Servo 2  Position7 Select Pb
OR        M02137	// Servo 2  Position7 Select'g
AND LOAD
AND NOT   M02106	// Servo 2  Position1 Select Pb
AND NOT   M02107	// Servo 2  Position2 Select Pb
AND NOT   M02108	// Servo 2  Position3 Select Pb
AND NOT   M02109	// Servo 2  Position4 Select Pb
AND NOT   M0210A	// Servo 2  Position5 Select Pb
AND NOT   M0210B	// Servo 2  Position6 Select Pb
AND NOT   M0210D	// Servo 2  Position8 Select Pb
OUT       M02137	// Servo 2  Position7 Select'g
; L124
LOAD      M02151	// Servo 2 수동선택
LOAD      M0210D	// Servo 2  Position8 Select Pb
OR        M02138	// Servo 2  Position8 Select'g
AND LOAD
AND NOT   M02106	// Servo 2  Position1 Select Pb
AND NOT   M02107	// Servo 2  Position2 Select Pb
AND NOT   M02108	// Servo 2  Position3 Select Pb
AND NOT   M02109	// Servo 2  Position4 Select Pb
AND NOT   M0210A	// Servo 2  Position5 Select Pb
AND NOT   M0210B	// Servo 2  Position6 Select Pb
AND NOT   M0210C	// Servo 2  Position7 Select Pb
OUT       M02138	// Servo 2  Position8 Select'g
; L126
LOAD      M02151	// Servo 2 수동선택
AND       M02131	// Servo 2  Position 1 Select'g
AND       D002211.C	// 서보 2 이동완료 (MEND)
LOADD=    D002250 D002214	// 서보 2 등록 포지션 1번 Low / 서보 2 Table 1 위치 데이타 Low
OR        F00093
AND LOAD
OUT       M02116	// Servo 2  Position1 Select Comple
; L128
LOAD      M02151	// Servo 2 수동선택
AND       M02132	// Servo 2  Position2 Select'g
AND       D002211.C	// 서보 2 이동완료 (MEND)
LOADD=    D002252 D002214	// 서보 2 등록 포지션 2번 Low / 서보 2 Table 1 위치 데이타 Low
OR        F00093
AND LOAD
OUT       M02117	// Servo 2  Position2 Select Comple

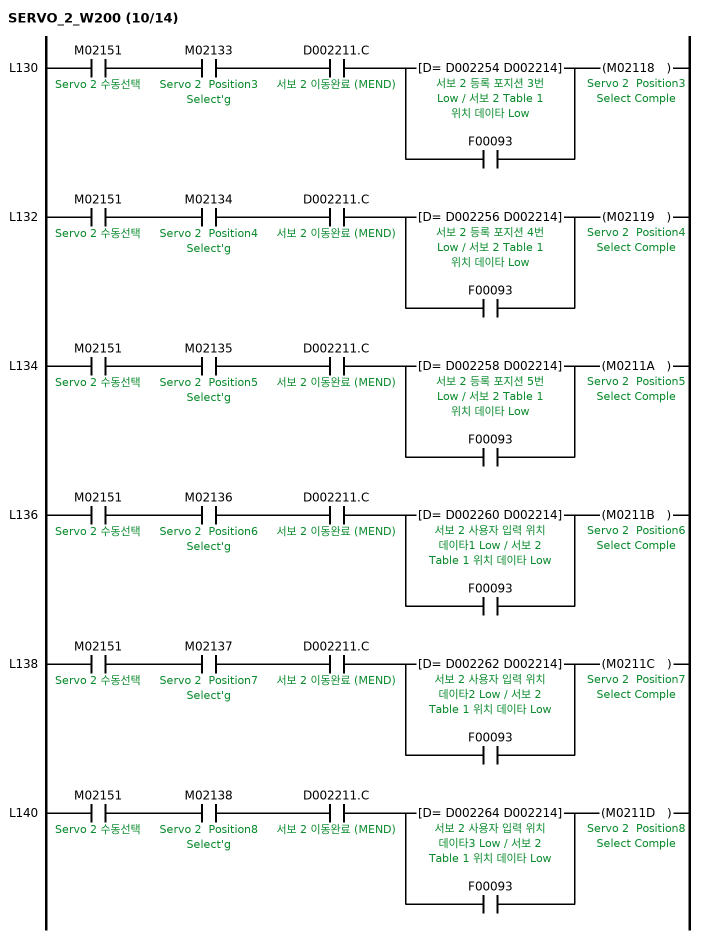
; L130
LOAD      M02151	// Servo 2 수동선택
AND       M02133	// Servo 2  Position3 Select'g
AND       D002211.C	// 서보 2 이동완료 (MEND)
LOADD=    D002254 D002214	// 서보 2 등록 포지션 3번 Low / 서보 2 Table 1 위치 데이타 Low
OR        F00093
AND LOAD
OUT       M02118	// Servo 2  Position3 Select Comple
; L132
LOAD      M02151	// Servo 2 수동선택
AND       M02134	// Servo 2  Position4 Select'g
AND       D002211.C	// 서보 2 이동완료 (MEND)
LOADD=    D002256 D002214	// 서보 2 등록 포지션 4번 Low / 서보 2 Table 1 위치 데이타 Low
OR        F00093
AND LOAD
OUT       M02119	// Servo 2  Position4 Select Comple
; L134
LOAD      M02151	// Servo 2 수동선택
AND       M02135	// Servo 2  Position5 Select'g
AND       D002211.C	// 서보 2 이동완료 (MEND)
LOADD=    D002258 D002214	// 서보 2 등록 포지션 5번 Low / 서보 2 Table 1 위치 데이타 Low
OR        F00093
AND LOAD
OUT       M0211A	// Servo 2  Position5 Select Comple
; L136
LOAD      M02151	// Servo 2 수동선택
AND       M02136	// Servo 2  Position6 Select'g
AND       D002211.C	// 서보 2 이동완료 (MEND)
LOADD=    D002260 D002214	// 서보 2 사용자 입력 위치 데이타1 Low / 서보 2 Table 1 위치 데이타 Low
OR        F00093
AND LOAD
OUT       M0211B	// Servo 2  Position6 Select Comple
; L138
LOAD      M02151	// Servo 2 수동선택
AND       M02137	// Servo 2  Position7 Select'g
AND       D002211.C	// 서보 2 이동완료 (MEND)
LOADD=    D002262 D002214	// 서보 2 사용자 입력 위치 데이타2 Low / 서보 2 Table 1 위치 데이타 Low
OR        F00093
AND LOAD
OUT       M0211C	// Servo 2  Position7 Select Comple
; L140
LOAD      M02151	// Servo 2 수동선택
AND       M02138	// Servo 2  Position8 Select'g
AND       D002211.C	// 서보 2 이동완료 (MEND)
LOADD=    D002264 D002214	// 서보 2 사용자 입력 위치 데이타3 Low / 서보 2 Table 1 위치 데이타 Low
OR        F00093
AND LOAD
OUT       M0211D	// Servo 2  Position8 Select Comple

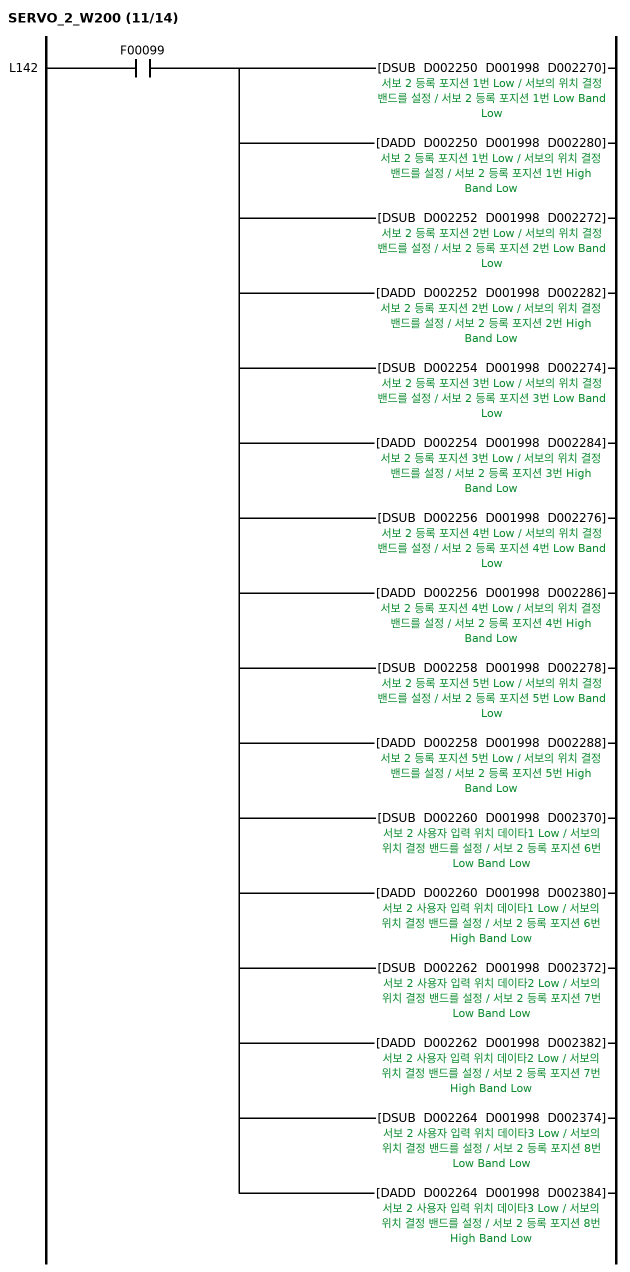
; L142
LOAD      F00099
DSUB      D002250 D001998 D002270	// 서보 2 등록 포지션 1번 Low / 서보의 위치 결정 밴드를 설정 / 서보 2 등록 포지션 1번 Low Band Low
DADD      D002250 D001998 D002280	// 서보 2 등록 포지션 1번 Low / 서보의 위치 결정 밴드를 설정 / 서보 2 등록 포지션 1번 High Band Low
DSUB      D002252 D001998 D002272	// 서보 2 등록 포지션 2번 Low / 서보의 위치 결정 밴드를 설정 / 서보 2 등록 포지션 2번 Low Band Low
DADD      D002252 D001998 D002282	// 서보 2 등록 포지션 2번 Low / 서보의 위치 결정 밴드를 설정 / 서보 2 등록 포지션 2번 High Band Low
DSUB      D002254 D001998 D002274	// 서보 2 등록 포지션 3번 Low / 서보의 위치 결정 밴드를 설정 / 서보 2 등록 포지션 3번 Low Band Low
DADD      D002254 D001998 D002284	// 서보 2 등록 포지션 3번 Low / 서보의 위치 결정 밴드를 설정 / 서보 2 등록 포지션 3번 High Band Low
DSUB      D002256 D001998 D002276	// 서보 2 등록 포지션 4번 Low / 서보의 위치 결정 밴드를 설정 / 서보 2 등록 포지션 4번 Low Band Low
DADD      D002256 D001998 D002286	// 서보 2 등록 포지션 4번 Low / 서보의 위치 결정 밴드를 설정 / 서보 2 등록 포지션 4번 High Band Low
DSUB      D002258 D001998 D002278	// 서보 2 등록 포지션 5번 Low / 서보의 위치 결정 밴드를 설정 / 서보 2 등록 포지션 5번 Low Band Low
DADD      D002258 D001998 D002288	// 서보 2 등록 포지션 5번 Low / 서보의 위치 결정 밴드를 설정 / 서보 2 등록 포지션 5번 High Band Low
DSUB      D002260 D001998 D002370	// 서보 2 사용자 입력 위치 데이타1 Low / 서보의 위치 결정 밴드를 설정 / 서보 2 등록 포지션 6번 Low Band Low
DADD      D002260 D001998 D002380	// 서보 2 사용자 입력 위치 데이타1 Low / 서보의 위치 결정 밴드를 설정 / 서보 2 등록 포지션 6번 High Band Low
DSUB      D002262 D001998 D002372	// 서보 2 사용자 입력 위치 데이타2 Low / 서보의 위치 결정 밴드를 설정 / 서보 2 등록 포지션 7번 Low Band Low
DADD      D002262 D001998 D002382	// 서보 2 사용자 입력 위치 데이타2 Low / 서보의 위치 결정 밴드를 설정 / 서보 2 등록 포지션 7번 High Band Low
DSUB      D002264 D001998 D002374	// 서보 2 사용자 입력 위치 데이타3 Low / 서보의 위치 결정 밴드를 설정 / 서보 2 등록 포지션 8번 Low Band Low
DADD      D002264 D001998 D002384	// 서보 2 사용자 입력 위치 데이타3 Low / 서보의 위치 결정 밴드를 설정 / 서보 2 등록 포지션 8번 High Band Low

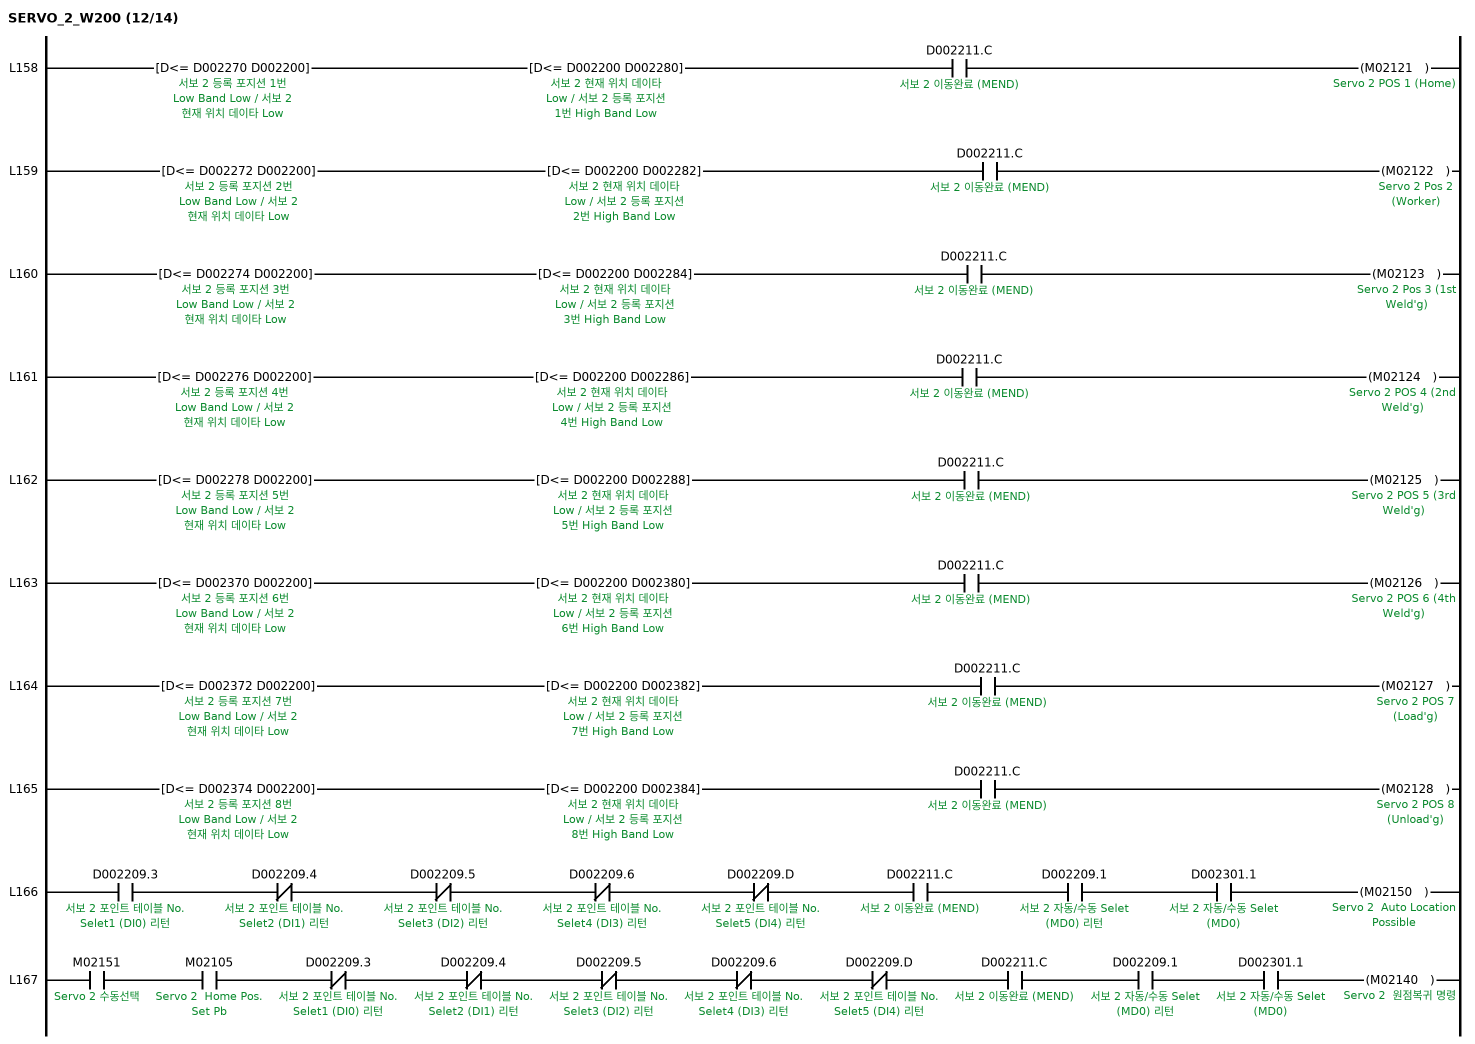
; L158
LOADD<=   D002270 D002200	// 서보 2 등록 포지션 1번 Low Band Low / 서보 2 현재 위치 데이타 Low
ANDD<=    D002200 D002280	// 서보 2 현재 위치 데이타 Low / 서보 2 등록 포지션 1번 High Band Low
AND       D002211.C	// 서보 2 이동완료 (MEND)
OUT       M02121	// Servo 2 POS 1 (Home)
; L159
LOADD<=   D002272 D002200	// 서보 2 등록 포지션 2번 Low Band Low / 서보 2 현재 위치 데이타 Low
ANDD<=    D002200 D002282	// 서보 2 현재 위치 데이타 Low / 서보 2 등록 포지션 2번 High Band Low
AND       D002211.C	// 서보 2 이동완료 (MEND)
OUT       M02122	// Servo 2 Pos 2 (Worker)
; L160
LOADD<=   D002274 D002200	// 서보 2 등록 포지션 3번 Low Band Low / 서보 2 현재 위치 데이타 Low
ANDD<=    D002200 D002284	// 서보 2 현재 위치 데이타 Low / 서보 2 등록 포지션 3번 High Band Low
AND       D002211.C	// 서보 2 이동완료 (MEND)
OUT       M02123	// Servo 2 Pos 3 (1st Weld'g)
; L161
LOADD<=   D002276 D002200	// 서보 2 등록 포지션 4번 Low Band Low / 서보 2 현재 위치 데이타 Low
ANDD<=    D002200 D002286	// 서보 2 현재 위치 데이타 Low / 서보 2 등록 포지션 4번 High Band Low
AND       D002211.C	// 서보 2 이동완료 (MEND)
OUT       M02124	// Servo 2 POS 4 (2nd Weld'g)
; L162
LOADD<=   D002278 D002200	// 서보 2 등록 포지션 5번 Low Band Low / 서보 2 현재 위치 데이타 Low
ANDD<=    D002200 D002288	// 서보 2 현재 위치 데이타 Low / 서보 2 등록 포지션 5번 High Band Low
AND       D002211.C	// 서보 2 이동완료 (MEND)
OUT       M02125	// Servo 2 POS 5 (3rd Weld'g)
; L163
LOADD<=   D002370 D002200	// 서보 2 등록 포지션 6번 Low Band Low / 서보 2 현재 위치 데이타 Low
ANDD<=    D002200 D002380	// 서보 2 현재 위치 데이타 Low / 서보 2 등록 포지션 6번 High Band Low
AND       D002211.C	// 서보 2 이동완료 (MEND)
OUT       M02126	// Servo 2 POS 6 (4th Weld'g)
; L164
LOADD<=   D002372 D002200	// 서보 2 등록 포지션 7번 Low Band Low / 서보 2 현재 위치 데이타 Low
ANDD<=    D002200 D002382	// 서보 2 현재 위치 데이타 Low / 서보 2 등록 포지션 7번 High Band Low
AND       D002211.C	// 서보 2 이동완료 (MEND)
OUT       M02127	// Servo 2 POS 7 (Load'g)
; L165
LOADD<=   D002374 D002200	// 서보 2 등록 포지션 8번 Low Band Low / 서보 2 현재 위치 데이타 Low
ANDD<=    D002200 D002384	// 서보 2 현재 위치 데이타 Low / 서보 2 등록 포지션 8번 High Band Low
AND       D002211.C	// 서보 2 이동완료 (MEND)
OUT       M02128	// Servo 2 POS 8 (Unload'g)
; L166
LOAD      D002209.3	// 서보 2 포인트 테이블 No. Selet1 (DI0) 리턴
AND NOT   D002209.4	// 서보 2 포인트 테이블 No. Selet2 (DI1) 리턴
AND NOT   D002209.5	// 서보 2 포인트 테이블 No. Selet3 (DI2) 리턴
AND NOT   D002209.6	// 서보 2 포인트 테이블 No. Selet4 (DI3) 리턴
AND NOT   D002209.D	// 서보 2 포인트 테이블 No. Selet5 (DI4) 리턴
AND       D002211.C	// 서보 2 이동완료 (MEND)
AND       D002209.1	// 서보 2 자동/수동 Selet (MD0) 리턴
AND       D002301.1	// 서보 2 자동/수동 Selet (MD0)
OUT       M02150	// Servo 2  Auto Location Possible
; L167
LOAD      M02151	// Servo 2 수동선택
AND       M02105	// Servo 2  Home Pos. Set Pb
AND NOT   D002209.3	// 서보 2 포인트 테이블 No. Selet1 (DI0) 리턴
AND NOT   D002209.4	// 서보 2 포인트 테이블 No. Selet2 (DI1) 리턴
AND NOT   D002209.5	// 서보 2 포인트 테이블 No. Selet3 (DI2) 리턴
AND NOT   D002209.6	// 서보 2 포인트 테이블 No. Selet4 (DI3) 리턴
AND NOT   D002209.D	// 서보 2 포인트 테이블 No. Selet5 (DI4) 리턴
AND       D002211.C	// 서보 2 이동완료 (MEND)
AND       D002209.1	// 서보 2 자동/수동 Selet (MD0) 리턴
AND       D002301.1	// 서보 2 자동/수동 Selet (MD0)
OUT       M02140	// Servo 2  원점복귀 명령

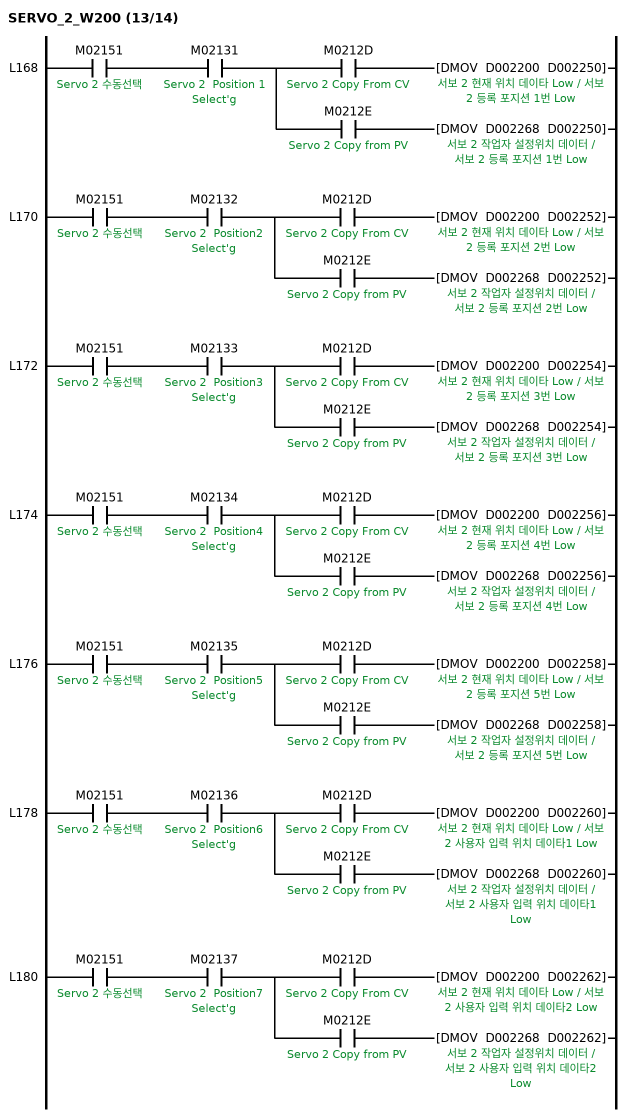
; L168
LOAD      M02151	// Servo 2 수동선택
AND       M02131	// Servo 2  Position 1 Select'g
MPUSH
AND       M0212D	// Servo 2 Copy From CV
DMOV      D002200 D002250	// 서보 2 현재 위치 데이타 Low / 서보 2 등록 포지션 1번 Low
MPOP
AND       M0212E	// Servo 2 Copy from PV
DMOV      D002268 D002250	// 서보 2 작업자 설정위치 데이터 / 서보 2 등록 포지션 1번 Low
; L170
LOAD      M02151	// Servo 2 수동선택
AND       M02132	// Servo 2  Position2 Select'g
MPUSH
AND       M0212D	// Servo 2 Copy From CV
DMOV      D002200 D002252	// 서보 2 현재 위치 데이타 Low / 서보 2 등록 포지션 2번 Low
MPOP
AND       M0212E	// Servo 2 Copy from PV
DMOV      D002268 D002252	// 서보 2 작업자 설정위치 데이터 / 서보 2 등록 포지션 2번 Low
; L172
LOAD      M02151	// Servo 2 수동선택
AND       M02133	// Servo 2  Position3 Select'g
MPUSH
AND       M0212D	// Servo 2 Copy From CV
DMOV      D002200 D002254	// 서보 2 현재 위치 데이타 Low / 서보 2 등록 포지션 3번 Low
MPOP
AND       M0212E	// Servo 2 Copy from PV
DMOV      D002268 D002254	// 서보 2 작업자 설정위치 데이터 / 서보 2 등록 포지션 3번 Low
; L174
LOAD      M02151	// Servo 2 수동선택
AND       M02134	// Servo 2  Position4 Select'g
MPUSH
AND       M0212D	// Servo 2 Copy From CV
DMOV      D002200 D002256	// 서보 2 현재 위치 데이타 Low / 서보 2 등록 포지션 4번 Low
MPOP
AND       M0212E	// Servo 2 Copy from PV
DMOV      D002268 D002256	// 서보 2 작업자 설정위치 데이터 / 서보 2 등록 포지션 4번 Low
; L176
LOAD      M02151	// Servo 2 수동선택
AND       M02135	// Servo 2  Position5 Select'g
MPUSH
AND       M0212D	// Servo 2 Copy From CV
DMOV      D002200 D002258	// 서보 2 현재 위치 데이타 Low / 서보 2 등록 포지션 5번 Low
MPOP
AND       M0212E	// Servo 2 Copy from PV
DMOV      D002268 D002258	// 서보 2 작업자 설정위치 데이터 / 서보 2 등록 포지션 5번 Low
; L178
LOAD      M02151	// Servo 2 수동선택
AND       M02136	// Servo 2  Position6 Select'g
MPUSH
AND       M0212D	// Servo 2 Copy From CV
DMOV      D002200 D002260	// 서보 2 현재 위치 데이타 Low / 서보 2 사용자 입력 위치 데이타1 Low
MPOP
AND       M0212E	// Servo 2 Copy from PV
DMOV      D002268 D002260	// 서보 2 작업자 설정위치 데이터 / 서보 2 사용자 입력 위치 데이타1 Low
; L180
LOAD      M02151	// Servo 2 수동선택
AND       M02137	// Servo 2  Position7 Select'g
MPUSH
AND       M0212D	// Servo 2 Copy From CV
DMOV      D002200 D002262	// 서보 2 현재 위치 데이타 Low / 서보 2 사용자 입력 위치 데이타2 Low
MPOP
AND       M0212E	// Servo 2 Copy from PV
DMOV      D002268 D002262	// 서보 2 작업자 설정위치 데이터 / 서보 2 사용자 입력 위치 데이타2 Low

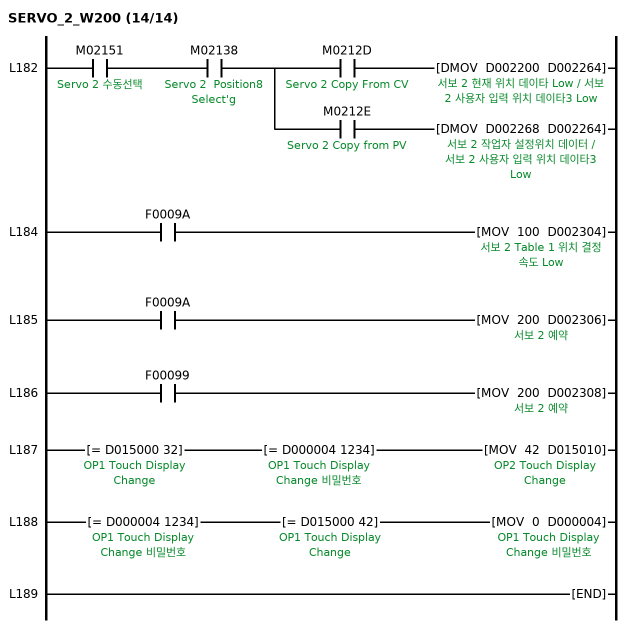
; L182
LOAD      M02151	// Servo 2 수동선택
AND       M02138	// Servo 2  Position8 Select'g
MPUSH
AND       M0212D	// Servo 2 Copy From CV
DMOV      D002200 D002264	// 서보 2 현재 위치 데이타 Low / 서보 2 사용자 입력 위치 데이타3 Low
MPOP
AND       M0212E	// Servo 2 Copy from PV
DMOV      D002268 D002264	// 서보 2 작업자 설정위치 데이터 / 서보 2 사용자 입력 위치 데이타3 Low
; L184
LOAD      F0009A
MOV       100 D002304	// 서보 2 Table 1 위치 결정 속도 Low
; L185
LOAD      F0009A
MOV       200 D002306	// 서보 2 예약
; L186
LOAD      F00099
MOV       200 D002308	// 서보 2 예약
; L187
LOAD=     D015000 32	// OP1 Touch Display Change
AND=      D000004 1234	// OP1 Touch Display Change 비밀번호
MOV       42 D015010	// OP2 Touch Display Change
; L188
LOAD=     D000004 1234	// OP1 Touch Display Change 비밀번호
AND=      D015000 42	// OP1 Touch Display Change
MOV       0 D000004	// OP1 Touch Display Change 비밀번호
; L189
END

PROGRAM SERVO_3_W400 (task: 스캔 프로그램)

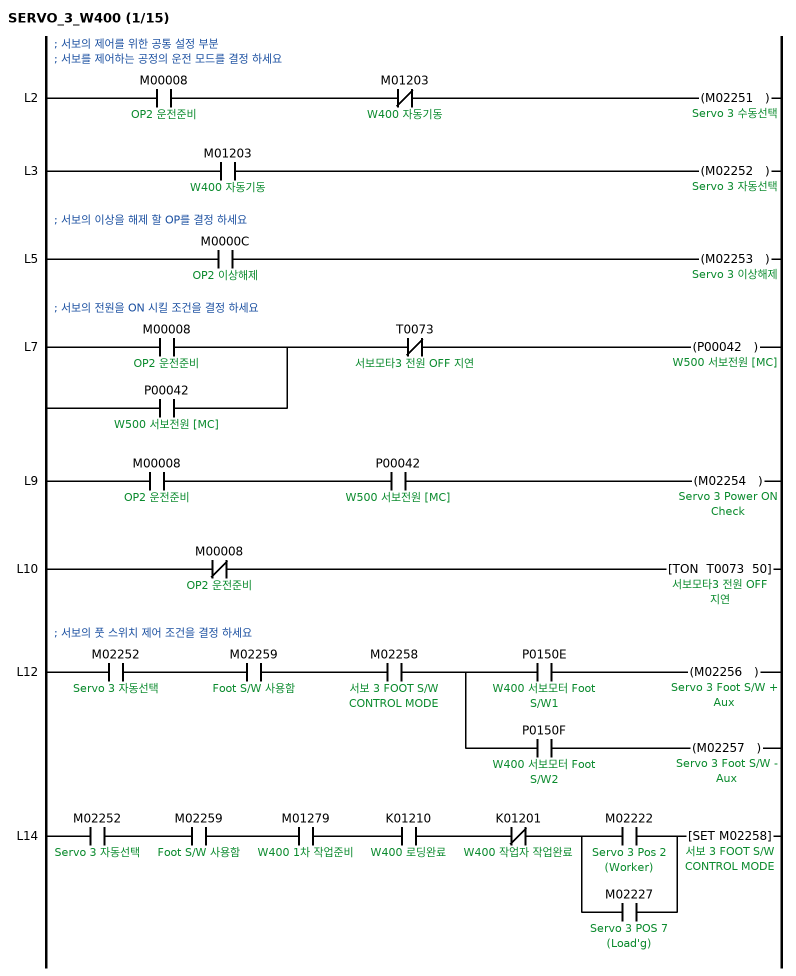
// 서보의 제어를 위한 공통 설정 부분
//     서보를 제어하는 공정의 운전 모드를 결정 하세요
; L2
LOAD      M00008	// OP2 운전준비
AND NOT   M01203	// W400 자동기동
OUT       M02251	// Servo 3 수동선택
; L3
LOAD      M01203	// W400 자동기동
OUT       M02252	// Servo 3 자동선택
//     서보의 이상을 해제 할 OP를 결정 하세요
; L5
LOAD      M0000C	// OP2 이상해제
OUT       M02253	// Servo 3 이상해제
//     서보의 전원을 ON 시킬 조건을 결정 하세요
; L7
LOAD      M00008	// OP2 운전준비
OR        P00042	// W500 서보전원 [MC]
AND NOT   T0073	// 서보모타3 전원 OFF 지연
OUT       P00042	// W500 서보전원 [MC]
; L9
LOAD      M00008	// OP2 운전준비
AND       P00042	// W500 서보전원 [MC]
OUT       M02254	// Servo 3 Power ON Check
; L10
LOAD NOT  M00008	// OP2 운전준비
TON       T0073 50	// 서보모타3 전원 OFF 지연
//     서보의 풋 스위치 제어 조건을 결정 하세요
; L12
LOAD      M02252	// Servo 3 자동선택
AND       M02259	// Foot S/W 사용함
AND       M02258	// 서보 3 FOOT S/W CONTROL MODE
MPUSH
AND       P0150E	// W400 서보모터 Foot S/W1
OUT       M02256	// Servo 3 Foot S/W + Aux
MPOP
AND       P0150F	// W400 서보모터 Foot S/W2
OUT       M02257	// Servo 3 Foot S/W - Aux
; L14
LOAD      M02252	// Servo 3 자동선택
AND       M02259	// Foot S/W 사용함
AND       M01279	// W400 1차 작업준비
AND       K01210	// W400 로딩완료
AND NOT   K01201	// W400 작업자 작업완료
LOAD      M02222	// Servo 3 Pos 2 (Worker)
OR        M02227	// Servo 3 POS 7 (Load'g)
AND LOAD
SET       M02258	// 서보 3 FOOT S/W CONTROL MODE

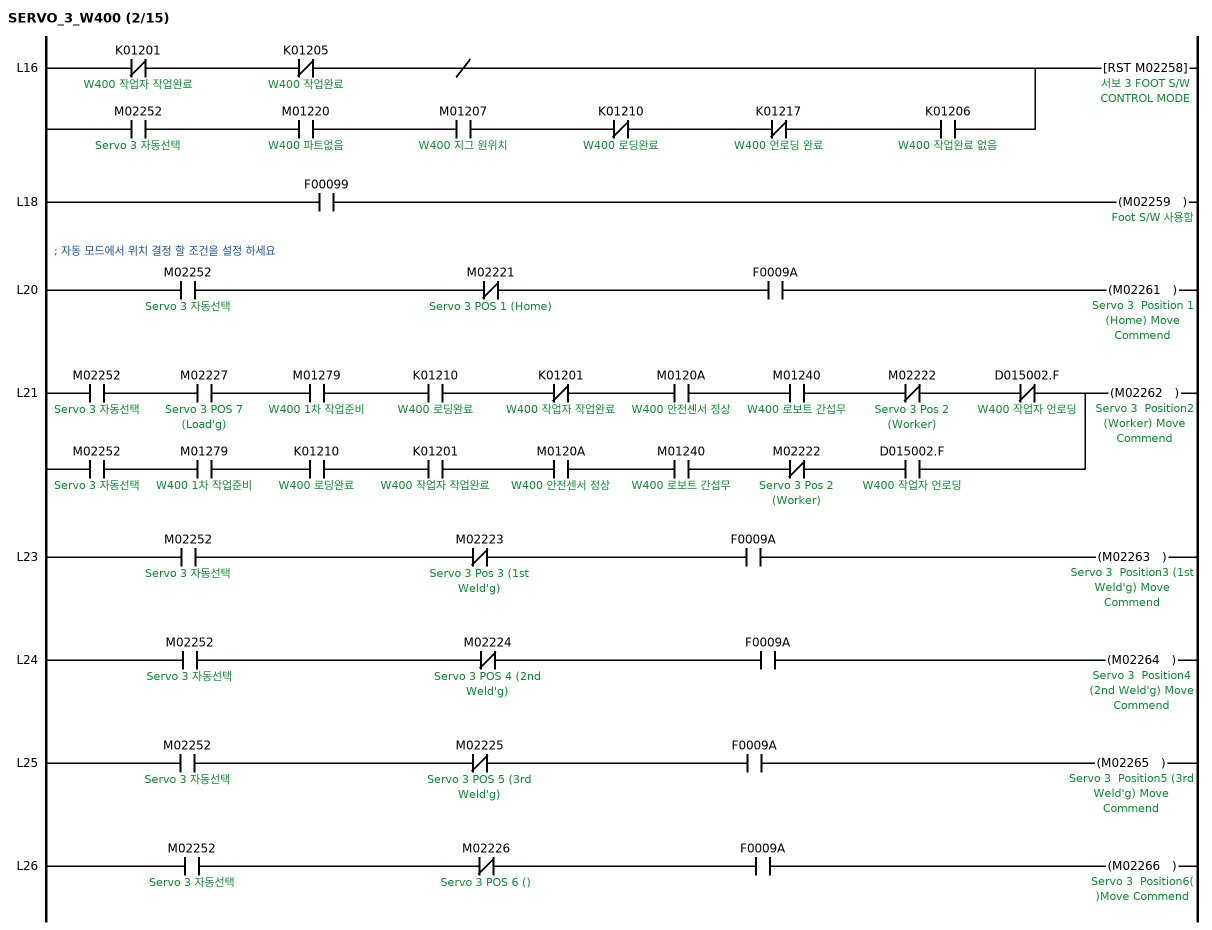
; L16
LOAD NOT  K01201	// W400 작업자 작업완료
AND NOT   K01205	// W400 작업완료
NOT
LOAD      M02252	// Servo 3 자동선택
AND       M01220	// W400 파트없음
AND       M01207	// W400 지그 원위치
AND NOT   K01210	// W400 로딩완료
AND NOT   K01217	// W400 언로딩 완료
AND       K01206	// W400 작업완료 없음
OR LOAD
RST       M02258	// 서보 3 FOOT S/W CONTROL MODE
; L18
LOAD      F00099
OUT       M02259	// Foot S/W 사용함
//     자동 모드에서 위치 결정 할 조건을 설정 하세요
; L20
LOAD      M02252	// Servo 3 자동선택
AND NOT   M02221	// Servo 3 POS 1 (Home)
AND       F0009A
OUT       M02261	// Servo 3  Position 1 (Home) Move Commend
; L21
LOAD      M02252	// Servo 3 자동선택
AND       M02227	// Servo 3 POS 7 (Load'g)
AND       M01279	// W400 1차 작업준비
AND       K01210	// W400 로딩완료
AND NOT   K01201	// W400 작업자 작업완료
AND       M0120A	// W400 안전센서 정상
AND       M01240	// W400 로보트 간섭무
AND NOT   M02222	// Servo 3 Pos 2 (Worker)
AND NOT   D015002.F	// W400 작업자 언로딩
LOAD      M02252	// Servo 3 자동선택
AND       M01279	// W400 1차 작업준비
AND       K01210	// W400 로딩완료
AND       K01201	// W400 작업자 작업완료
AND       M0120A	// W400 안전센서 정상
AND       M01240	// W400 로보트 간섭무
AND NOT   M02222	// Servo 3 Pos 2 (Worker)
AND       D015002.F	// W400 작업자 언로딩
OR LOAD
OUT       M02262	// Servo 3  Position2 (Worker) Move Commend
; L23
LOAD      M02252	// Servo 3 자동선택
AND NOT   M02223	// Servo 3 Pos 3 (1st Weld'g)
AND       F0009A
OUT       M02263	// Servo 3  Position3 (1st Weld'g) Move Commend
; L24
LOAD      M02252	// Servo 3 자동선택
AND NOT   M02224	// Servo 3 POS 4 (2nd Weld'g)
AND       F0009A
OUT       M02264	// Servo 3  Position4 (2nd Weld'g) Move Commend
; L25
LOAD      M02252	// Servo 3 자동선택
AND NOT   M02225	// Servo 3 POS 5 (3rd Weld'g)
AND       F0009A
OUT       M02265	// Servo 3  Position5 (3rd Weld'g) Move Commend
; L26
LOAD      M02252	// Servo 3 자동선택
AND NOT   M02226	// Servo 3 POS 6 ()
AND       F0009A
OUT       M02266	// Servo 3  Position6()Move Commend

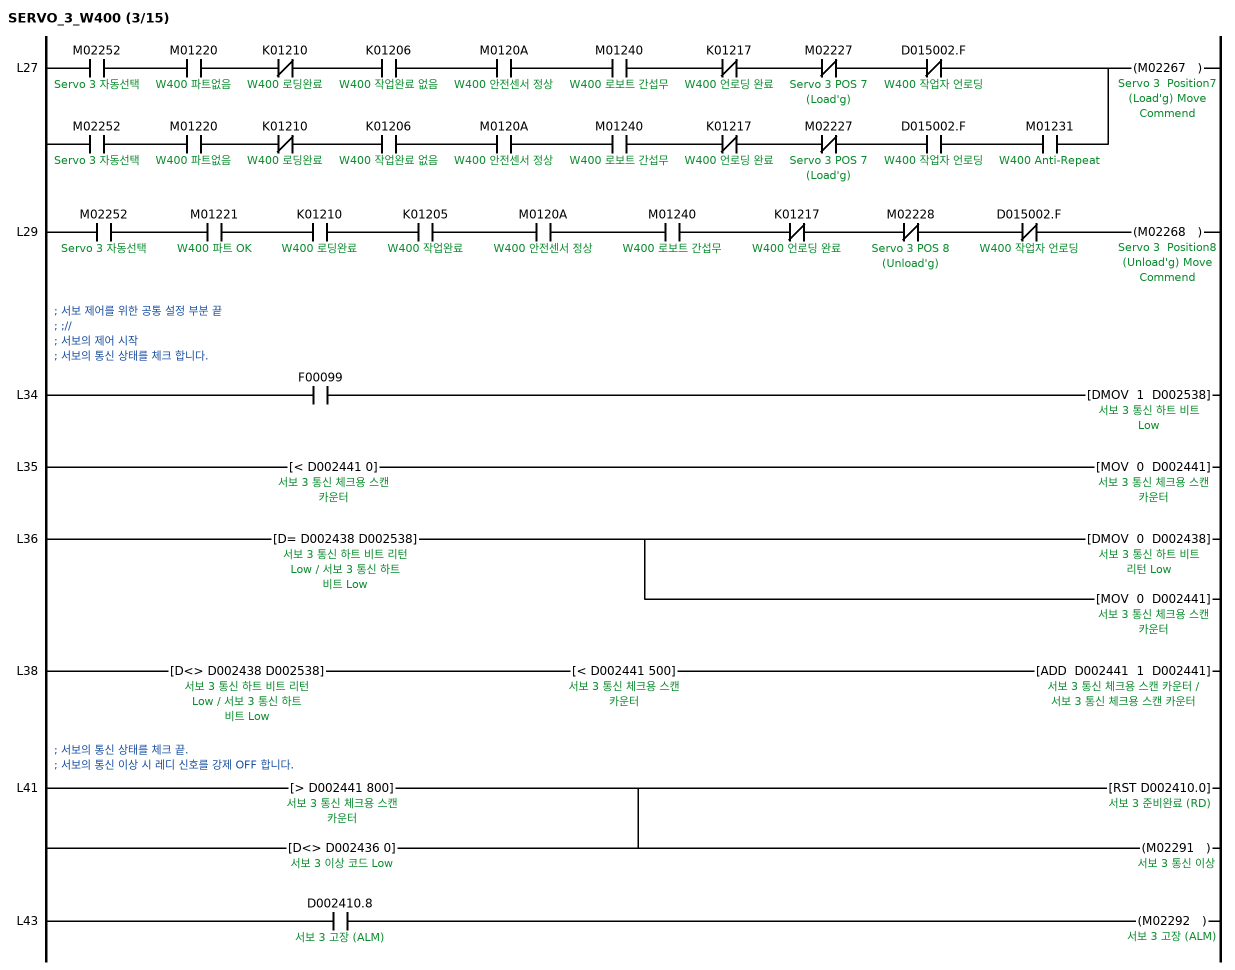
; L27
LOAD      M02252	// Servo 3 자동선택
AND       M01220	// W400 파트없음
AND NOT   K01210	// W400 로딩완료
AND       K01206	// W400 작업완료 없음
AND       M0120A	// W400 안전센서 정상
AND       M01240	// W400 로보트 간섭무
AND NOT   K01217	// W400 언로딩 완료
AND NOT   M02227	// Servo 3 POS 7 (Load'g)
AND NOT   D015002.F	// W400 작업자 언로딩
LOAD      M02252	// Servo 3 자동선택
AND       M01220	// W400 파트없음
AND NOT   K01210	// W400 로딩완료
AND       K01206	// W400 작업완료 없음
AND       M0120A	// W400 안전센서 정상
AND       M01240	// W400 로보트 간섭무
AND NOT   K01217	// W400 언로딩 완료
AND NOT   M02227	// Servo 3 POS 7 (Load'g)
AND       D015002.F	// W400 작업자 언로딩
AND       M01231	// W400 Anti-Repeat
OR LOAD
OUT       M02267	// Servo 3  Position7 (Load'g) Move Commend
; L29
LOAD      M02252	// Servo 3 자동선택
AND       M01221	// W400 파트 OK
AND       K01210	// W400 로딩완료
AND       K01205	// W400 작업완료
AND       M0120A	// W400 안전센서 정상
AND       M01240	// W400 로보트 간섭무
AND NOT   K01217	// W400 언로딩 완료
AND NOT   M02228	// Servo 3 POS 8 (Unload'g)
AND NOT   D015002.F	// W400 작업자 언로딩
OUT       M02268	// Servo 3  Position8 (Unload'g) Move Commend
// 서보 제어를 위한 공통 설정 부분 끝
// ;//
// 서보의 제어 시작
//     서보의 통신 상태를 체크 합니다.
; L34
LOAD      F00099
DMOV      1 D002538	// 서보 3 통신 하트 비트 Low
; L35
LOAD<     D002441 0	// 서보 3 통신 체크용 스캔 카운터
MOV       0 D002441	// 서보 3 통신 체크용 스캔 카운터
; L36
LOADD=    D002438 D002538	// 서보 3 통신 하트 비트 리턴 Low / 서보 3 통신 하트 비트 Low
DMOV      0 D002438	// 서보 3 통신 하트 비트 리턴 Low
MOV       0 D002441	// 서보 3 통신 체크용 스캔 카운터
; L38
LOADD<>   D002438 D002538	// 서보 3 통신 하트 비트 리턴 Low / 서보 3 통신 하트 비트 Low
AND<      D002441 500	// 서보 3 통신 체크용 스캔 카운터
ADD       D002441 1 D002441	// 서보 3 통신 체크용 스캔 카운터 / 서보 3 통신 체크용 스캔 카운터
//     서보의 통신 상태를 체크 끝.
//     서보의 통신 이상 시 레디 신호를 강제 OFF 합니다.
; L41
LOAD>     D002441 800	// 서보 3 통신 체크용 스캔 카운터
ORD<>     D002436 0	// 서보 3 이상 코드 Low
RST       D002410.0	// 서보 3 준비완료 (RD)
OUT       M02291	// 서보 3 통신 이상
; L43
LOAD      D002410.8	// 서보 3 고장 (ALM)
OUT       M02292	// 서보 3 고장 (ALM)

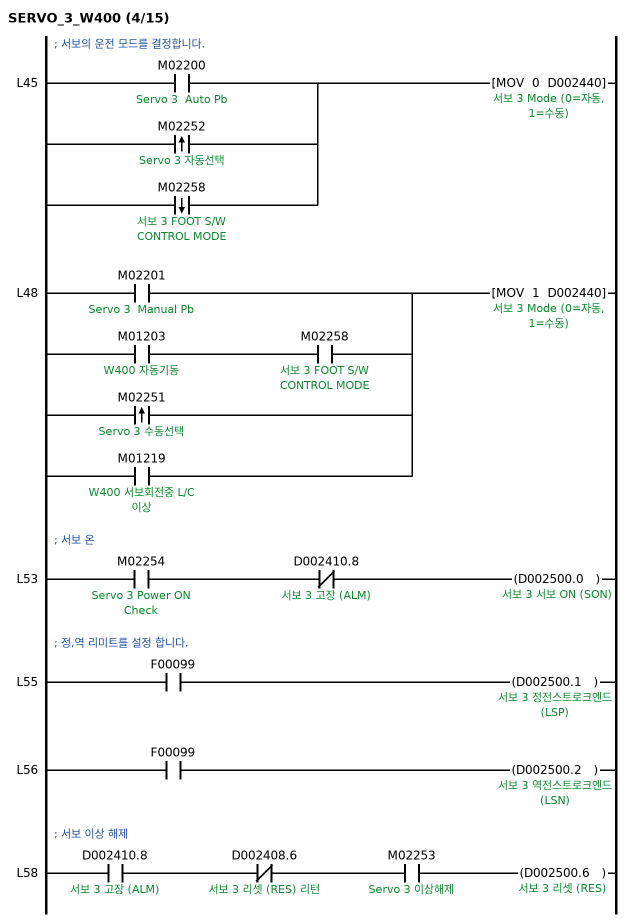
//     서보의 운전 모드를 결정합니다.
; L45
LOAD      M02200	// Servo 3  Auto Pb
ORP       M02252	// Servo 3 자동선택
ORN       M02258	// 서보 3 FOOT S/W CONTROL MODE
MOV       0 D002440	// 서보 3 Mode (0=자동, 1=수동)
; L48
LOAD      M02201	// Servo 3  Manual Pb
LOAD      M01203	// W400 자동기동
AND       M02258	// 서보 3 FOOT S/W CONTROL MODE
OR LOAD
ORP       M02251	// Servo 3 수동선택
OR        M01219	// W400 서보회전중 L/C 이상
MOV       1 D002440	// 서보 3 Mode (0=자동, 1=수동)
//     서보 온
; L53
LOAD      M02254	// Servo 3 Power ON Check
AND NOT   D002410.8	// 서보 3 고장 (ALM)
OUT       D002500.0	// 서보 3 서보 ON (SON)
//     정,역 리미트를 설정 합니다.
; L55
LOAD      F00099
OUT       D002500.1	// 서보 3 정전스트로크엔드 (LSP)
; L56
LOAD      F00099
OUT       D002500.2	// 서보 3 역전스트로크엔드 (LSN)
//     서보 이상 해제
; L58
LOAD      D002410.8	// 서보 3 고장 (ALM)
AND NOT   D002408.6	// 서보 3 리셋 (RES) 리턴
AND       M02253	// Servo 3 이상해제
OUT       D002500.6	// 서보 3 리셋 (RES)

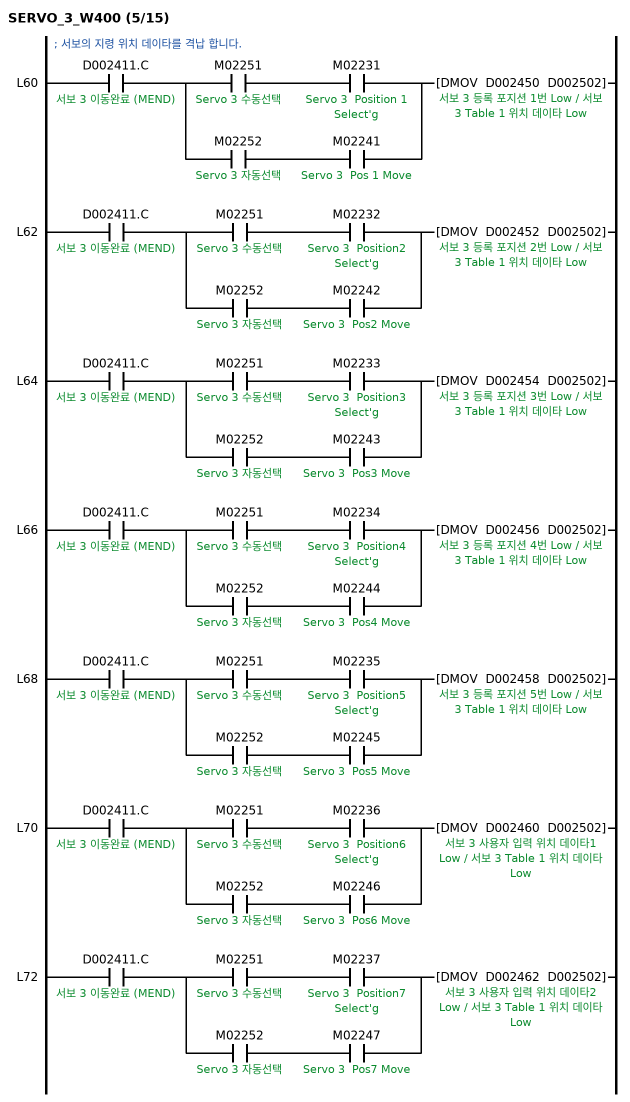
//     서보의 지령 위치 데이타를 격납 합니다.
; L60
LOAD      D002411.C	// 서보 3 이동완료 (MEND)
LOAD      M02251	// Servo 3 수동선택
AND       M02231	// Servo 3  Position 1 Select'g
LOAD      M02252	// Servo 3 자동선택
AND       M02241	// Servo 3  Pos 1 Move
OR LOAD
AND LOAD
DMOV      D002450 D002502	// 서보 3 등록 포지션 1번 Low / 서보 3 Table 1 위치 데이타 Low
; L62
LOAD      D002411.C	// 서보 3 이동완료 (MEND)
LOAD      M02251	// Servo 3 수동선택
AND       M02232	// Servo 3  Position2 Select'g
LOAD      M02252	// Servo 3 자동선택
AND       M02242	// Servo 3  Pos2 Move
OR LOAD
AND LOAD
DMOV      D002452 D002502	// 서보 3 등록 포지션 2번 Low / 서보 3 Table 1 위치 데이타 Low
; L64
LOAD      D002411.C	// 서보 3 이동완료 (MEND)
LOAD      M02251	// Servo 3 수동선택
AND       M02233	// Servo 3  Position3 Select'g
LOAD      M02252	// Servo 3 자동선택
AND       M02243	// Servo 3  Pos3 Move
OR LOAD
AND LOAD
DMOV      D002454 D002502	// 서보 3 등록 포지션 3번 Low / 서보 3 Table 1 위치 데이타 Low
; L66
LOAD      D002411.C	// 서보 3 이동완료 (MEND)
LOAD      M02251	// Servo 3 수동선택
AND       M02234	// Servo 3  Position4 Select'g
LOAD      M02252	// Servo 3 자동선택
AND       M02244	// Servo 3  Pos4 Move
OR LOAD
AND LOAD
DMOV      D002456 D002502	// 서보 3 등록 포지션 4번 Low / 서보 3 Table 1 위치 데이타 Low
; L68
LOAD      D002411.C	// 서보 3 이동완료 (MEND)
LOAD      M02251	// Servo 3 수동선택
AND       M02235	// Servo 3  Position5 Select'g
LOAD      M02252	// Servo 3 자동선택
AND       M02245	// Servo 3  Pos5 Move
OR LOAD
AND LOAD
DMOV      D002458 D002502	// 서보 3 등록 포지션 5번 Low / 서보 3 Table 1 위치 데이타 Low
; L70
LOAD      D002411.C	// 서보 3 이동완료 (MEND)
LOAD      M02251	// Servo 3 수동선택
AND       M02236	// Servo 3  Position6 Select'g
LOAD      M02252	// Servo 3 자동선택
AND       M02246	// Servo 3  Pos6 Move
OR LOAD
AND LOAD
DMOV      D002460 D002502	// 서보 3 사용자 입력 위치 데이타1 Low / 서보 3 Table 1 위치 데이타 Low
; L72
LOAD      D002411.C	// 서보 3 이동완료 (MEND)
LOAD      M02251	// Servo 3 수동선택
AND       M02237	// Servo 3  Position7 Select'g
LOAD      M02252	// Servo 3 자동선택
AND       M02247	// Servo 3  Pos7 Move
OR LOAD
AND LOAD
DMOV      D002462 D002502	// 서보 3 사용자 입력 위치 데이타2 Low / 서보 3 Table 1 위치 데이타 Low

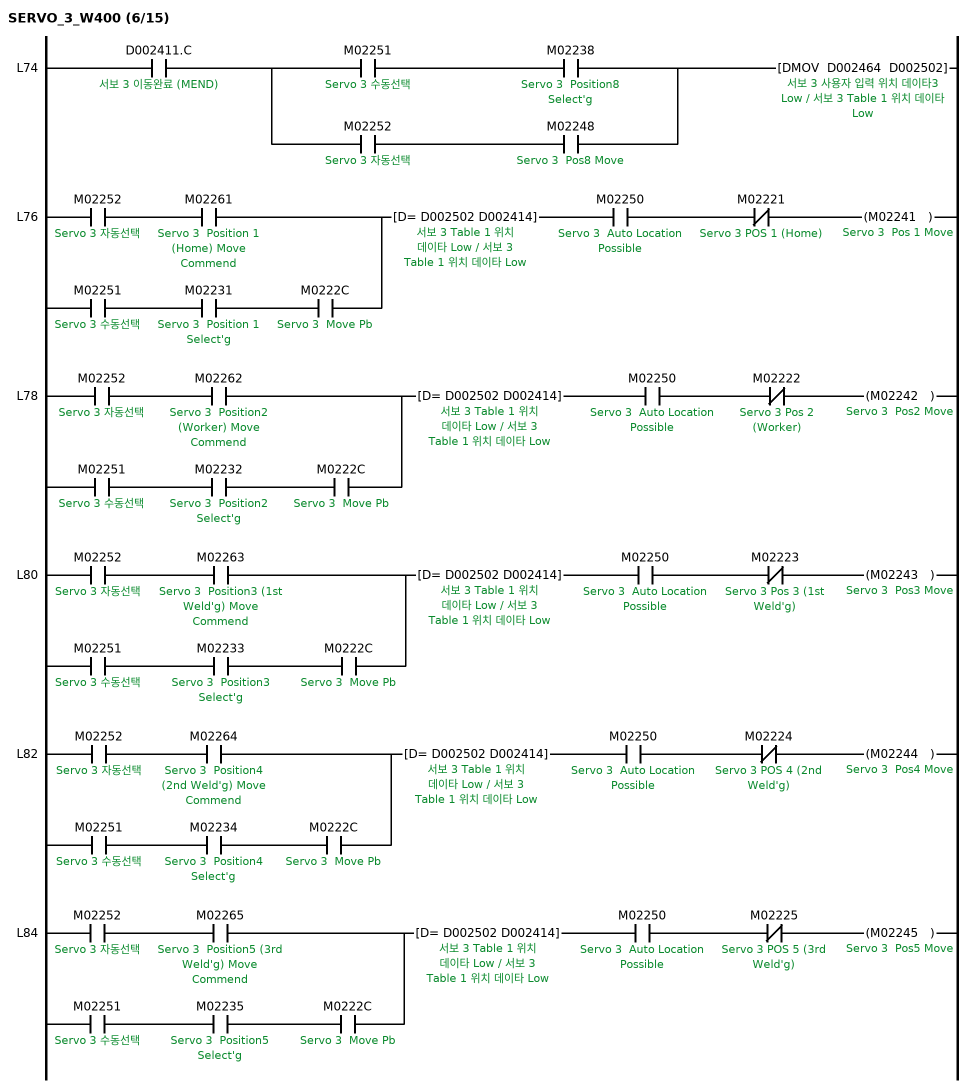
; L74
LOAD      D002411.C	// 서보 3 이동완료 (MEND)
LOAD      M02251	// Servo 3 수동선택
AND       M02238	// Servo 3  Position8 Select'g
LOAD      M02252	// Servo 3 자동선택
AND       M02248	// Servo 3  Pos8 Move
OR LOAD
AND LOAD
DMOV      D002464 D002502	// 서보 3 사용자 입력 위치 데이타3 Low / 서보 3 Table 1 위치 데이타 Low
; L76
LOAD      M02252	// Servo 3 자동선택
AND       M02261	// Servo 3  Position 1 (Home) Move Commend
LOAD      M02251	// Servo 3 수동선택
AND       M02231	// Servo 3  Position 1 Select'g
AND       M0222C	// Servo 3  Move Pb
OR LOAD
ANDD=     D002502 D002414	// 서보 3 Table 1 위치 데이타 Low / 서보 3 Table 1 위치 데이타 Low
AND       M02250	// Servo 3  Auto Location Possible
AND NOT   M02221	// Servo 3 POS 1 (Home)
OUT       M02241	// Servo 3  Pos 1 Move
; L78
LOAD      M02252	// Servo 3 자동선택
AND       M02262	// Servo 3  Position2 (Worker) Move Commend
LOAD      M02251	// Servo 3 수동선택
AND       M02232	// Servo 3  Position2 Select'g
AND       M0222C	// Servo 3  Move Pb
OR LOAD
ANDD=     D002502 D002414	// 서보 3 Table 1 위치 데이타 Low / 서보 3 Table 1 위치 데이타 Low
AND       M02250	// Servo 3  Auto Location Possible
AND NOT   M02222	// Servo 3 Pos 2 (Worker)
OUT       M02242	// Servo 3  Pos2 Move
; L80
LOAD      M02252	// Servo 3 자동선택
AND       M02263	// Servo 3  Position3 (1st Weld'g) Move Commend
LOAD      M02251	// Servo 3 수동선택
AND       M02233	// Servo 3  Position3 Select'g
AND       M0222C	// Servo 3  Move Pb
OR LOAD
ANDD=     D002502 D002414	// 서보 3 Table 1 위치 데이타 Low / 서보 3 Table 1 위치 데이타 Low
AND       M02250	// Servo 3  Auto Location Possible
AND NOT   M02223	// Servo 3 Pos 3 (1st Weld'g)
OUT       M02243	// Servo 3  Pos3 Move
; L82
LOAD      M02252	// Servo 3 자동선택
AND       M02264	// Servo 3  Position4 (2nd Weld'g) Move Commend
LOAD      M02251	// Servo 3 수동선택
AND       M02234	// Servo 3  Position4 Select'g
AND       M0222C	// Servo 3  Move Pb
OR LOAD
ANDD=     D002502 D002414	// 서보 3 Table 1 위치 데이타 Low / 서보 3 Table 1 위치 데이타 Low
AND       M02250	// Servo 3  Auto Location Possible
AND NOT   M02224	// Servo 3 POS 4 (2nd Weld'g)
OUT       M02244	// Servo 3  Pos4 Move
; L84
LOAD      M02252	// Servo 3 자동선택
AND       M02265	// Servo 3  Position5 (3rd Weld'g) Move Commend
LOAD      M02251	// Servo 3 수동선택
AND       M02235	// Servo 3  Position5 Select'g
AND       M0222C	// Servo 3  Move Pb
OR LOAD
ANDD=     D002502 D002414	// 서보 3 Table 1 위치 데이타 Low / 서보 3 Table 1 위치 데이타 Low
AND       M02250	// Servo 3  Auto Location Possible
AND NOT   M02225	// Servo 3 POS 5 (3rd Weld'g)
OUT       M02245	// Servo 3  Pos5 Move

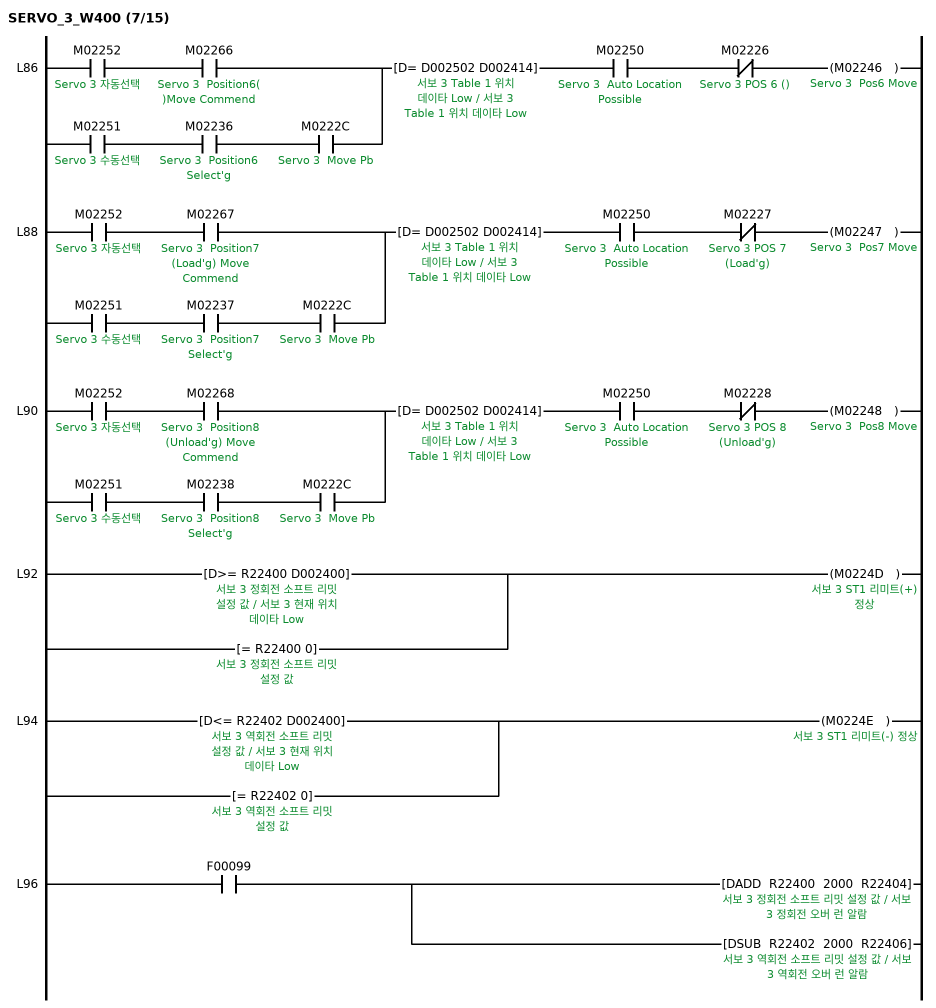
; L86
LOAD      M02252	// Servo 3 자동선택
AND       M02266	// Servo 3  Position6()Move Commend
LOAD      M02251	// Servo 3 수동선택
AND       M02236	// Servo 3  Position6 Select'g
AND       M0222C	// Servo 3  Move Pb
OR LOAD
ANDD=     D002502 D002414	// 서보 3 Table 1 위치 데이타 Low / 서보 3 Table 1 위치 데이타 Low
AND       M02250	// Servo 3  Auto Location Possible
AND NOT   M02226	// Servo 3 POS 6 ()
OUT       M02246	// Servo 3  Pos6 Move
; L88
LOAD      M02252	// Servo 3 자동선택
AND       M02267	// Servo 3  Position7 (Load'g) Move Commend
LOAD      M02251	// Servo 3 수동선택
AND       M02237	// Servo 3  Position7 Select'g
AND       M0222C	// Servo 3  Move Pb
OR LOAD
ANDD=     D002502 D002414	// 서보 3 Table 1 위치 데이타 Low / 서보 3 Table 1 위치 데이타 Low
AND       M02250	// Servo 3  Auto Location Possible
AND NOT   M02227	// Servo 3 POS 7 (Load'g)
OUT       M02247	// Servo 3  Pos7 Move
; L90
LOAD      M02252	// Servo 3 자동선택
AND       M02268	// Servo 3  Position8 (Unload'g) Move Commend
LOAD      M02251	// Servo 3 수동선택
AND       M02238	// Servo 3  Position8 Select'g
AND       M0222C	// Servo 3  Move Pb
OR LOAD
ANDD=     D002502 D002414	// 서보 3 Table 1 위치 데이타 Low / 서보 3 Table 1 위치 데이타 Low
AND       M02250	// Servo 3  Auto Location Possible
AND NOT   M02228	// Servo 3 POS 8 (Unload'g)
OUT       M02248	// Servo 3  Pos8 Move
; L92
LOADD>=   R22400 D002400	// 서보 3 정회전 소프트 리밋 설정 값 / 서보 3 현재 위치 데이타 Low
OR=       R22400 0	// 서보 3 정회전 소프트 리밋 설정 값
OUT       M0224D	// 서보 3 ST1 리미트(+) 정상
; L94
LOADD<=   R22402 D002400	// 서보 3 역회전 소프트 리밋 설정 값 / 서보 3 현재 위치 데이타 Low
OR=       R22402 0	// 서보 3 역회전 소프트 리밋 설정 값
OUT       M0224E	// 서보 3 ST1 리미트(-) 정상
; L96
LOAD      F00099
DADD      R22400 2000 R22404	// 서보 3 정회전 소프트 리밋 설정 값 / 서보 3 정회전 오버 런 알람
DSUB      R22402 2000 R22406	// 서보 3 역회전 소프트 리밋 설정 값 / 서보 3 역회전 오버 런 알람

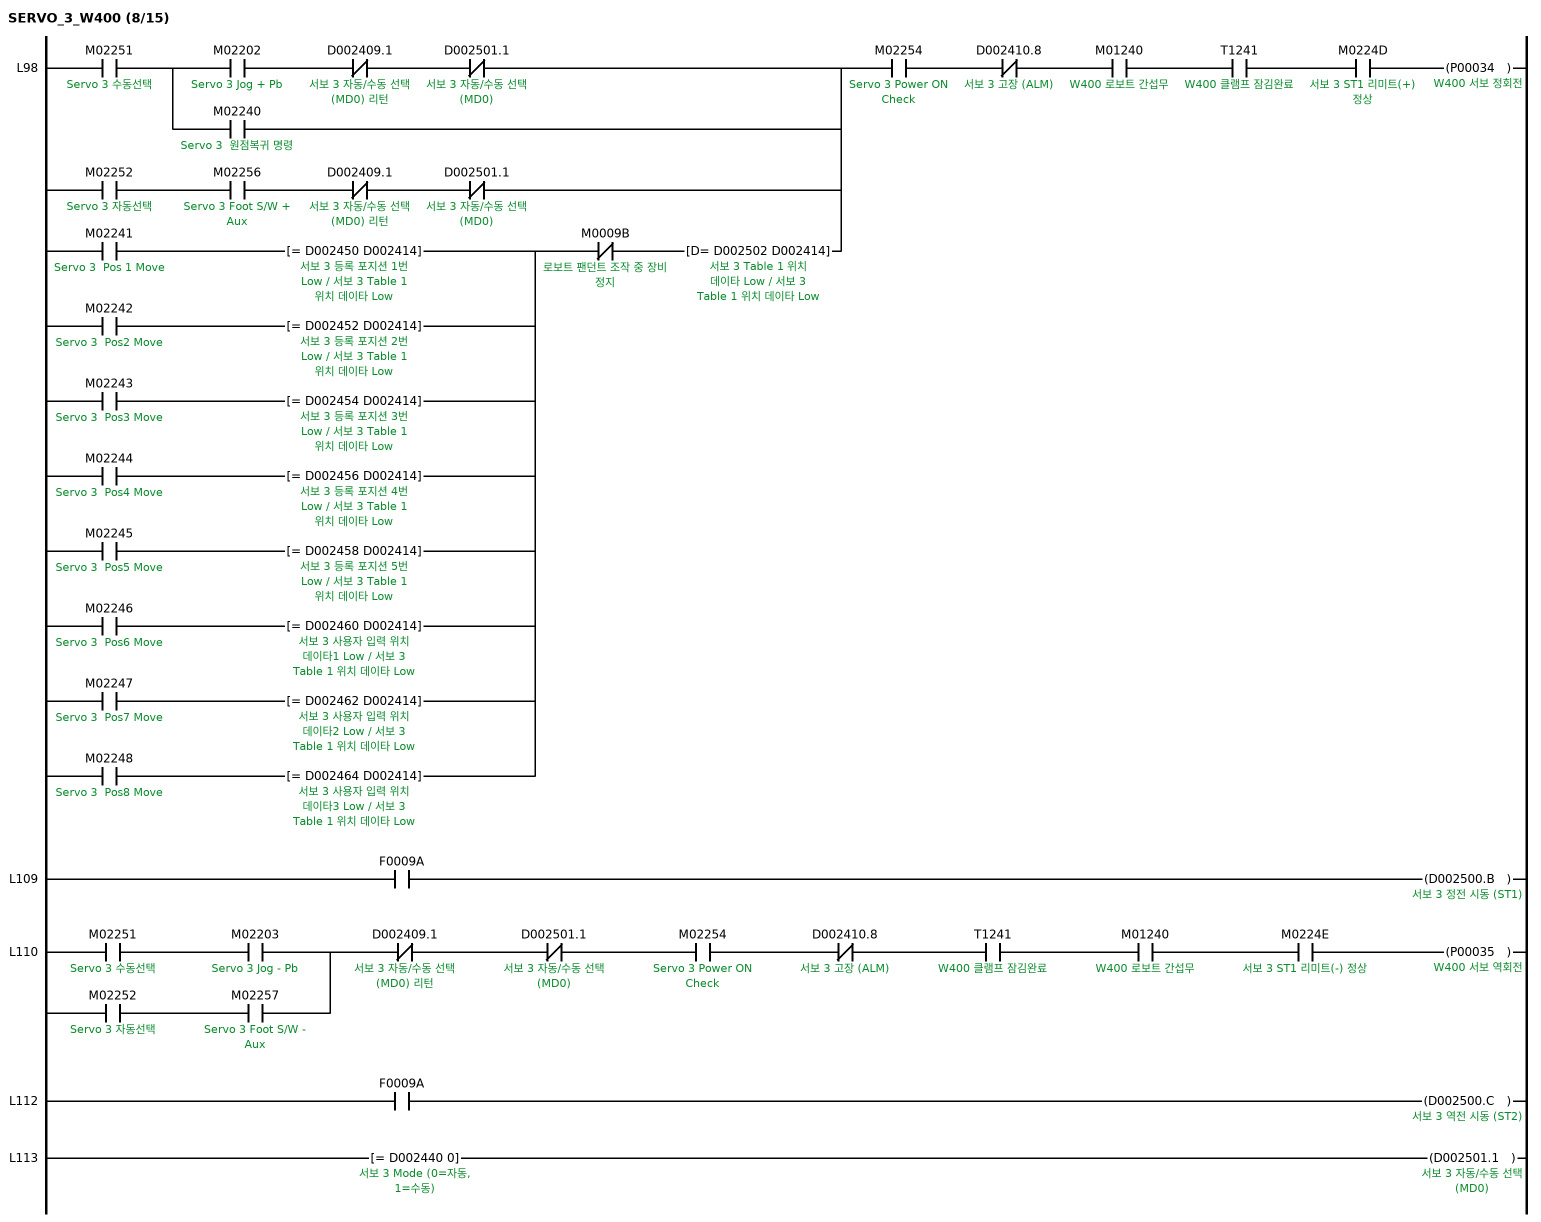
; L98
LOAD      M02251	// Servo 3 수동선택
LOAD      M02202	// Servo 3 Jog + Pb
AND NOT   D002409.1	// 서보 3 자동/수동 선택 (MD0) 리턴
AND NOT   D002501.1	// 서보 3 자동/수동 선택 (MD0)
OR        M02240	// Servo 3  원점복귀 명령
AND LOAD
LOAD      M02252	// Servo 3 자동선택
AND       M02256	// Servo 3 Foot S/W + Aux
AND NOT   D002409.1	// 서보 3 자동/수동 선택 (MD0) 리턴
AND NOT   D002501.1	// 서보 3 자동/수동 선택 (MD0)
OR LOAD
LOAD      M02241	// Servo 3  Pos 1 Move
AND=      D002450 D002414	// 서보 3 등록 포지션 1번 Low / 서보 3 Table 1 위치 데이타 Low
LOAD      M02242	// Servo 3  Pos2 Move
AND=      D002452 D002414	// 서보 3 등록 포지션 2번 Low / 서보 3 Table 1 위치 데이타 Low
OR LOAD
LOAD      M02243	// Servo 3  Pos3 Move
AND=      D002454 D002414	// 서보 3 등록 포지션 3번 Low / 서보 3 Table 1 위치 데이타 Low
OR LOAD
LOAD      M02244	// Servo 3  Pos4 Move
AND=      D002456 D002414	// 서보 3 등록 포지션 4번 Low / 서보 3 Table 1 위치 데이타 Low
OR LOAD
LOAD      M02245	// Servo 3  Pos5 Move
AND=      D002458 D002414	// 서보 3 등록 포지션 5번 Low / 서보 3 Table 1 위치 데이타 Low
OR LOAD
LOAD      M02246	// Servo 3  Pos6 Move
AND=      D002460 D002414	// 서보 3 사용자 입력 위치 데이타1 Low / 서보 3 Table 1 위치 데이타 Low
OR LOAD
LOAD      M02247	// Servo 3  Pos7 Move
AND=      D002462 D002414	// 서보 3 사용자 입력 위치 데이타2 Low / 서보 3 Table 1 위치 데이타 Low
OR LOAD
LOAD      M02248	// Servo 3  Pos8 Move
AND=      D002464 D002414	// 서보 3 사용자 입력 위치 데이타3 Low / 서보 3 Table 1 위치 데이타 Low
OR LOAD
AND NOT   M0009B	// 로보트 팬던트 조작 중 장비 정지
ANDD=     D002502 D002414	// 서보 3 Table 1 위치 데이타 Low / 서보 3 Table 1 위치 데이타 Low
OR LOAD
AND       M02254	// Servo 3 Power ON Check
AND NOT   D002410.8	// 서보 3 고장 (ALM)
AND       M01240	// W400 로보트 간섭무
AND       T1241	// W400 클램프 잠김완료
AND       M0224D	// 서보 3 ST1 리미트(+) 정상
OUT       P00034	// W400 서보 정회전
; L109
LOAD      F0009A
OUT       D002500.B	// 서보 3 정전 시동 (ST1)
; L110
LOAD      M02251	// Servo 3 수동선택
AND       M02203	// Servo 3 Jog - Pb
LOAD      M02252	// Servo 3 자동선택
AND       M02257	// Servo 3 Foot S/W - Aux
OR LOAD
AND NOT   D002409.1	// 서보 3 자동/수동 선택 (MD0) 리턴
AND NOT   D002501.1	// 서보 3 자동/수동 선택 (MD0)
AND       M02254	// Servo 3 Power ON Check
AND NOT   D002410.8	// 서보 3 고장 (ALM)
AND       T1241	// W400 클램프 잠김완료
AND       M01240	// W400 로보트 간섭무
AND       M0224E	// 서보 3 ST1 리미트(-) 정상
OUT       P00035	// W400 서보 역회전
; L112
LOAD      F0009A
OUT       D002500.C	// 서보 3 역전 시동 (ST2)
; L113
LOAD=     D002440 0	// 서보 3 Mode (0=자동, 1=수동)
OUT       D002501.1	// 서보 3 자동/수동 선택 (MD0)

